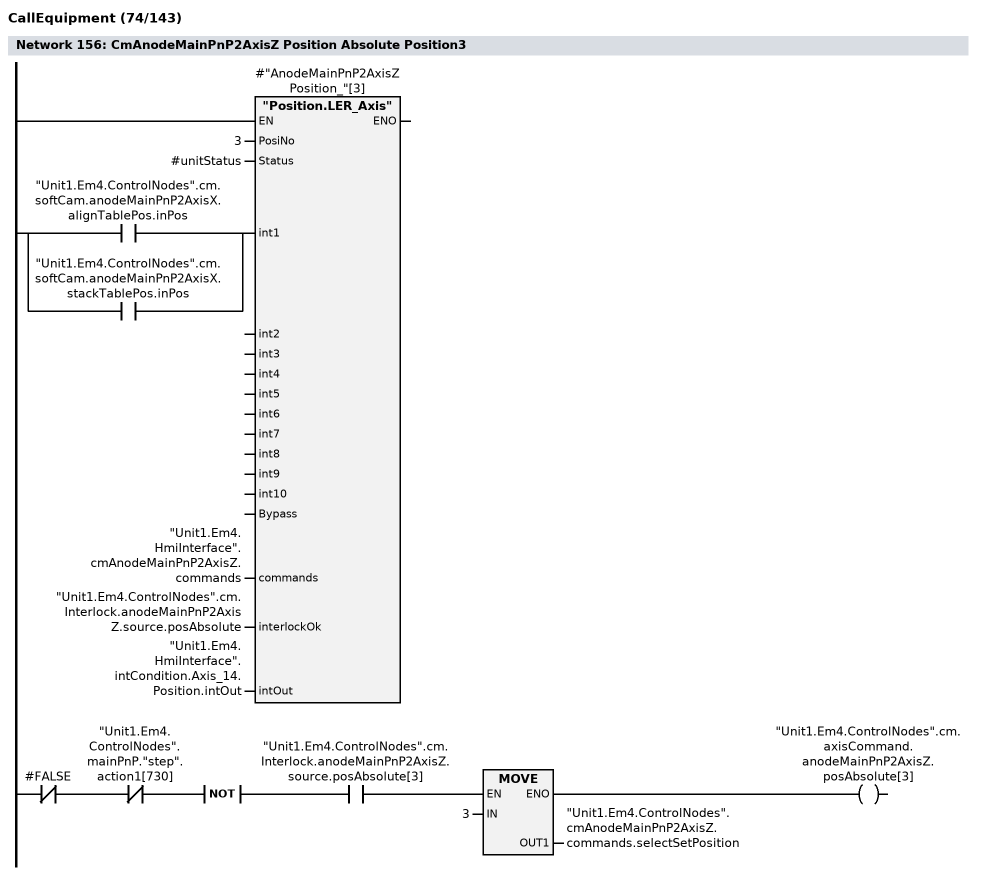
   RUNG wire#powerrail
      #"AnodeMainPnP2AxisZ Position_"[3](int1 := wire#w1, PosiNo := 3, Status := #unitStatus, int2 :=, int3 :=, int4 :=, int5 :=, int6 :=, int7 :=, int8 :=, int9 :=, int10 :=, Bypass :=, commands := "Unit1.Em4.HmiInterface".cmAnodeMainPnP2AxisZ.commands, interlockOk := "Unit1.Em4.ControlNodes".cm.Interlock.anodeMainPnP2AxisZ.source.posAbsolute, intOut := "Unit1.Em4.HmiInterface".intCondition.Axis_14.Position.intOut)
   END_RUNG
   RUNG wire#powerrail
      Contact( "Unit1.Em4.ControlNodes".cm.softCam.anodeMainPnP2AxisX.alignTablePos.inPos )
   END_RUNG wire#w1
   RUNG wire#powerrail
      Contact( "Unit1.Em4.ControlNodes".cm.softCam.anodeMainPnP2AxisX.stackTablePos.inPos )
   END_RUNG wire#w1
   RUNG wire#powerrail
      I_Contact( #FALSE )
      I_Contact( "Unit1.Em4.ControlNodes".mainPnP."step".action1[730] )
      Not()
      Contact( "Unit1.Em4.ControlNodes".cm.Interlock.anodeMainPnP2AxisZ.source.posAbsolute[3] )
      Move(in := 3, out1 => "Unit1.Em4.ControlNodes".cmAnodeMainPnP2AxisZ.commands.selectSetPosition)
      Coil( "Unit1.Em4.ControlNodes".cm.axisCommand.anodeMainPnP2AxisZ.posAbsolute[3] )
   END_RUNG
   // the same network as SCL:
   #"AnodeMainPnP2AxisZ Position_"[3](PosiNo := 3,   // "Position.LER_Axis"
                           Status := #unitStatus,
                           int1 := "Unit1.Em4.ControlNodes".cm.softCam.anodeMainPnP2AxisX.alignTablePos.inPos OR "Unit1.Em4.ControlNodes".cm.softCam.anodeMainPnP2AxisX.stackTablePos.inPos,
                           commands := "Unit1.Em4.HmiInterface".cmAnodeMainPnP2AxisZ.commands,
                           interlockOk := "Unit1.Em4.ControlNodes".cm.Interlock.anodeMainPnP2AxisZ.source.posAbsolute,
                           intOut := "Unit1.Em4.HmiInterface".intCondition.Axis_14.Position.intOut);
   #_w1 := NOT (NOT #FALSE AND NOT "Unit1.Em4.ControlNodes".mainPnP."step".action1[730]) AND "Unit1.Em4.ControlNodes".cm.Interlock.anodeMainPnP2AxisZ.source.posAbsolute[3];
   IF #_w1 THEN "Unit1.Em4.ControlNodes".cmAnodeMainPnP2AxisZ.commands.selectSetPosition := 3; END_IF;
   "Unit1.Em4.ControlNodes".cm.axisCommand.anodeMainPnP2AxisZ.posAbsolute[3] := #_w1;
END_REGION

REGION Network 157: CmAnodeMainPnP2AxisZ Position Absolute Position4
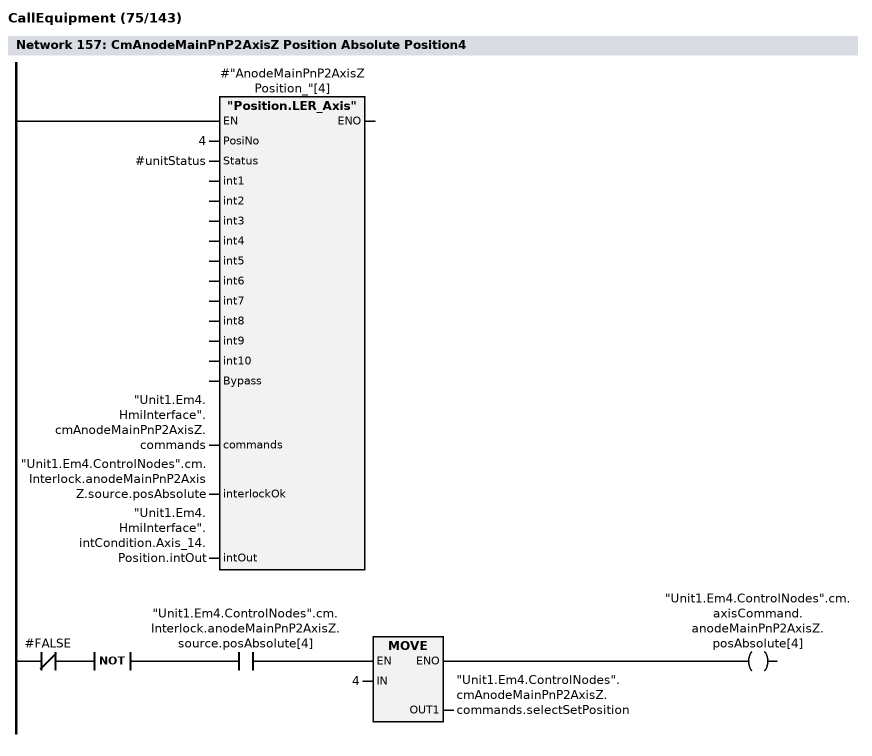
   RUNG wire#powerrail
      #"AnodeMainPnP2AxisZ Position_"[4](PosiNo := 4, Status := #unitStatus, int1 :=, int2 :=, int3 :=, int4 :=, int5 :=, int6 :=, int7 :=, int8 :=, int9 :=, int10 :=, Bypass :=, commands := "Unit1.Em4.HmiInterface".cmAnodeMainPnP2AxisZ.commands, interlockOk := "Unit1.Em4.ControlNodes".cm.Interlock.anodeMainPnP2AxisZ.source.posAbsolute, intOut := "Unit1.Em4.HmiInterface".intCondition.Axis_14.Position.intOut)
   END_RUNG
   RUNG wire#powerrail
      I_Contact( #FALSE )
      Not()
      Contact( "Unit1.Em4.ControlNodes".cm.Interlock.anodeMainPnP2AxisZ.source.posAbsolute[4] )
      Move(in := 4, out1 => "Unit1.Em4.ControlNodes".cmAnodeMainPnP2AxisZ.commands.selectSetPosition)
      Coil( "Unit1.Em4.ControlNodes".cm.axisCommand.anodeMainPnP2AxisZ.posAbsolute[4] )
   END_RUNG
   // the same network as SCL:
   #"AnodeMainPnP2AxisZ Position_"[4](PosiNo := 4,   // "Position.LER_Axis"
                           Status := #unitStatus,
                           commands := "Unit1.Em4.HmiInterface".cmAnodeMainPnP2AxisZ.commands,
                           interlockOk := "Unit1.Em4.ControlNodes".cm.Interlock.anodeMainPnP2AxisZ.source.posAbsolute,
                           intOut := "Unit1.Em4.HmiInterface".intCondition.Axis_14.Position.intOut);
   #_w1 := NOT (NOT #FALSE) AND "Unit1.Em4.ControlNodes".cm.Interlock.anodeMainPnP2AxisZ.source.posAbsolute[4];
   IF #_w1 THEN "Unit1.Em4.ControlNodes".cmAnodeMainPnP2AxisZ.commands.selectSetPosition := 4; END_IF;
   "Unit1.Em4.ControlNodes".cm.axisCommand.anodeMainPnP2AxisZ.posAbsolute[4] := #_w1;
END_REGION

REGION Network 158: CmAnodeMainPnP2AxisZ Position Absolute Position5
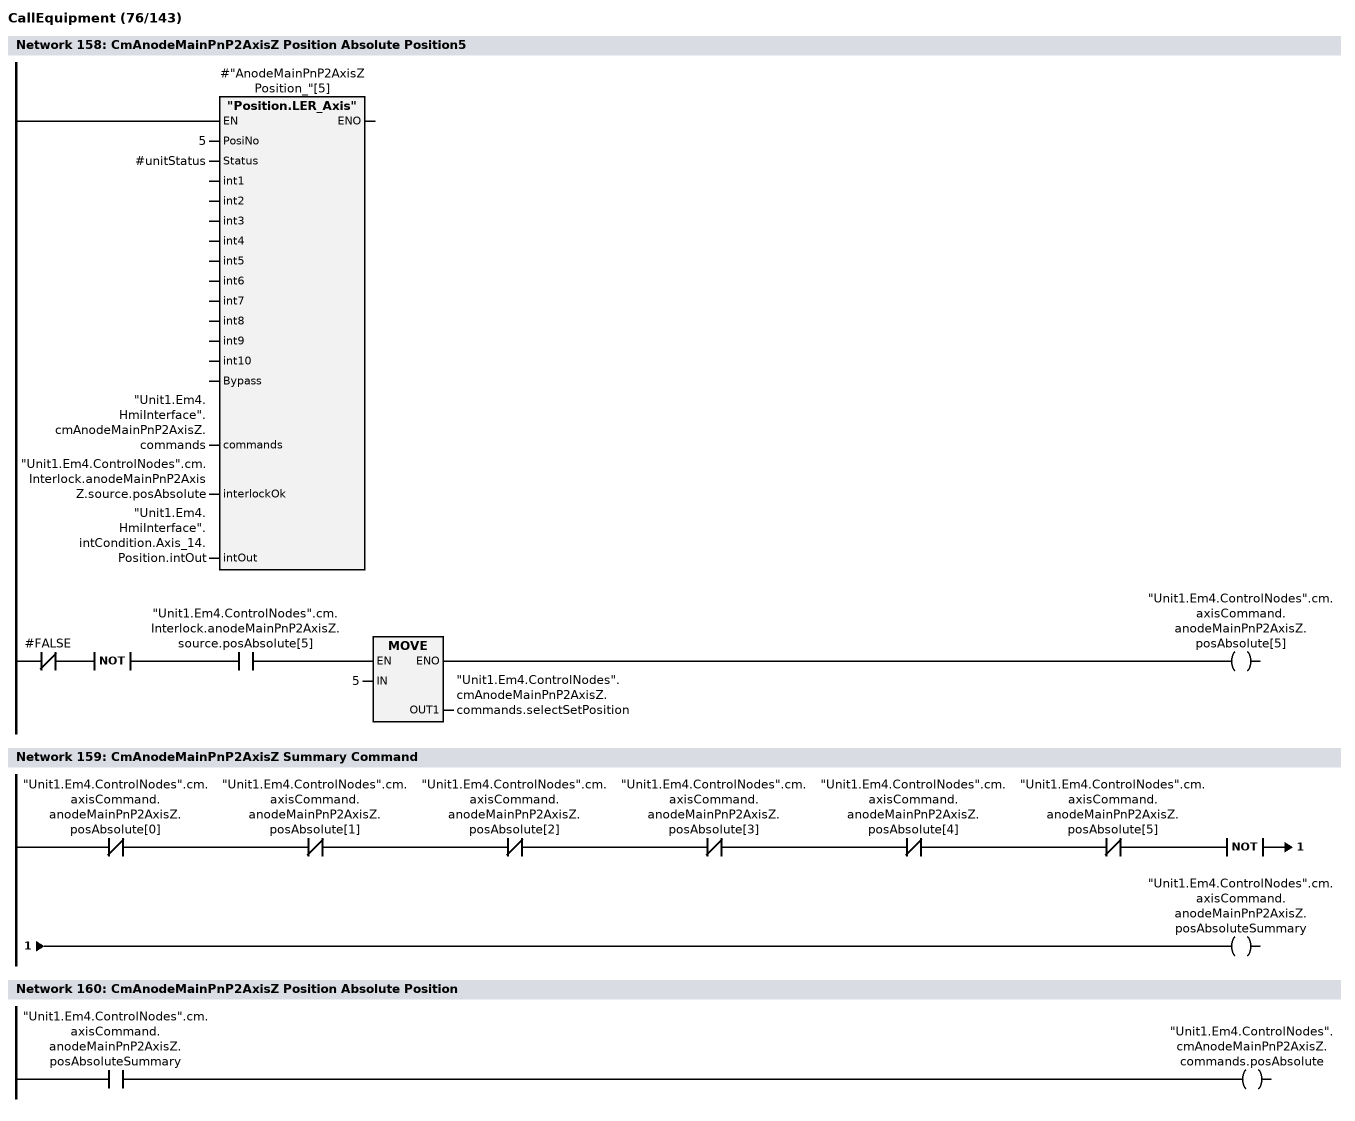
   RUNG wire#powerrail
      #"AnodeMainPnP2AxisZ Position_"[5](PosiNo := 5, Status := #unitStatus, int1 :=, int2 :=, int3 :=, int4 :=, int5 :=, int6 :=, int7 :=, int8 :=, int9 :=, int10 :=, Bypass :=, commands := "Unit1.Em4.HmiInterface".cmAnodeMainPnP2AxisZ.commands, interlockOk := "Unit1.Em4.ControlNodes".cm.Interlock.anodeMainPnP2AxisZ.source.posAbsolute, intOut := "Unit1.Em4.HmiInterface".intCondition.Axis_14.Position.intOut)
   END_RUNG
   RUNG wire#powerrail
      I_Contact( #FALSE )
      Not()
      Contact( "Unit1.Em4.ControlNodes".cm.Interlock.anodeMainPnP2AxisZ.source.posAbsolute[5] )
      Move(in := 5, out1 => "Unit1.Em4.ControlNodes".cmAnodeMainPnP2AxisZ.commands.selectSetPosition)
      Coil( "Unit1.Em4.ControlNodes".cm.axisCommand.anodeMainPnP2AxisZ.posAbsolute[5] )
   END_RUNG
   // the same network as SCL:
   #"AnodeMainPnP2AxisZ Position_"[5](PosiNo := 5,   // "Position.LER_Axis"
                           Status := #unitStatus,
                           commands := "Unit1.Em4.HmiInterface".cmAnodeMainPnP2AxisZ.commands,
                           interlockOk := "Unit1.Em4.ControlNodes".cm.Interlock.anodeMainPnP2AxisZ.source.posAbsolute,
                           intOut := "Unit1.Em4.HmiInterface".intCondition.Axis_14.Position.intOut);
   #_w1 := NOT (NOT #FALSE) AND "Unit1.Em4.ControlNodes".cm.Interlock.anodeMainPnP2AxisZ.source.posAbsolute[5];
   IF #_w1 THEN "Unit1.Em4.ControlNodes".cmAnodeMainPnP2AxisZ.commands.selectSetPosition := 5; END_IF;
   "Unit1.Em4.ControlNodes".cm.axisCommand.anodeMainPnP2AxisZ.posAbsolute[5] := #_w1;
END_REGION

REGION Network 159: CmAnodeMainPnP2AxisZ Summary Command
   RUNG wire#powerrail
      I_Contact( "Unit1.Em4.ControlNodes".cm.axisCommand.anodeMainPnP2AxisZ.posAbsolute[0] )
      I_Contact( "Unit1.Em4.ControlNodes".cm.axisCommand.anodeMainPnP2AxisZ.posAbsolute[1] )
      I_Contact( "Unit1.Em4.ControlNodes".cm.axisCommand.anodeMainPnP2AxisZ.posAbsolute[2] )
      I_Contact( "Unit1.Em4.ControlNodes".cm.axisCommand.anodeMainPnP2AxisZ.posAbsolute[3] )
      I_Contact( "Unit1.Em4.ControlNodes".cm.axisCommand.anodeMainPnP2AxisZ.posAbsolute[4] )
      I_Contact( "Unit1.Em4.ControlNodes".cm.axisCommand.anodeMainPnP2AxisZ.posAbsolute[5] )
      Not()
      Coil( "Unit1.Em4.ControlNodes".cm.axisCommand.anodeMainPnP2AxisZ.posAbsoluteSummary )
   END_RUNG
   // the same network as SCL:
   "Unit1.Em4.ControlNodes".cm.axisCommand.anodeMainPnP2AxisZ.posAbsoluteSummary := NOT (NOT "Unit1.Em4.ControlNodes".cm.axisCommand.anodeMainPnP2AxisZ.posAbsolute[0] AND NOT "Unit1.Em4.ControlNodes".cm.axisCommand.anodeMainPnP2AxisZ.posAbsolute[1] AND NOT "Unit1.Em4.ControlNodes".cm.axisCommand.anodeMainPnP2AxisZ.posAbsolute[2] AND NOT "Unit1.Em4.ControlNodes".cm.axisCommand.anodeMainPnP2AxisZ.posAbsolute[3] AND NOT "Unit1.Em4.ControlNodes".cm.axisCommand.anodeMainPnP2AxisZ.posAbsolute[4] AND NOT "Unit1.Em4.ControlNodes".cm.axisCommand.anodeMainPnP2AxisZ.posAbsolute[5]);
END_REGION

REGION Network 160: CmAnodeMainPnP2AxisZ Position Absolute Position
   RUNG wire#powerrail
      Contact( "Unit1.Em4.ControlNodes".cm.axisCommand.anodeMainPnP2AxisZ.posAbsoluteSummary )
      Coil( "Unit1.Em4.ControlNodes".cmAnodeMainPnP2AxisZ.commands.posAbsolute )
   END_RUNG
   // the same network as SCL:
   "Unit1.Em4.ControlNodes".cmAnodeMainPnP2AxisZ.commands.posAbsolute := "Unit1.Em4.ControlNodes".cm.axisCommand.anodeMainPnP2AxisZ.posAbsoluteSummary;
END_REGION

REGION Network 161: CmAnodeMainPnP1AxisZ Interlock Summary
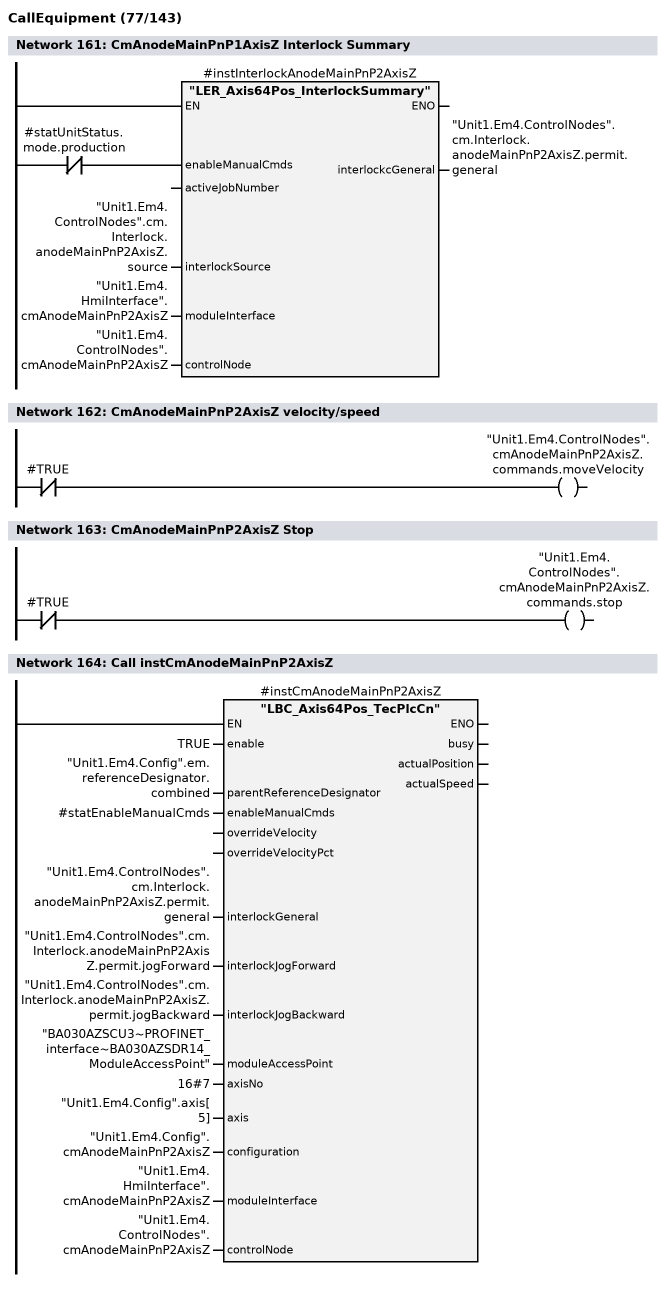
   RUNG wire#powerrail
      #instInterlockAnodeMainPnP2AxisZ(enableManualCmds := wire#w1, activeJobNumber :=, interlockSource := "Unit1.Em4.ControlNodes".cm.Interlock.anodeMainPnP2AxisZ.source, moduleInterface := "Unit1.Em4.HmiInterface".cmAnodeMainPnP2AxisZ, controlNode := "Unit1.Em4.ControlNodes".cmAnodeMainPnP2AxisZ, interlockcGeneral => "Unit1.Em4.ControlNodes".cm.Interlock.anodeMainPnP2AxisZ.permit.general)
   END_RUNG
   RUNG wire#powerrail
      I_Contact( #statUnitStatus.mode.production )
   END_RUNG wire#w1
   // the same network as SCL:
   #instInterlockAnodeMainPnP2AxisZ(enableManualCmds := NOT #statUnitStatus.mode.production,   // "LER_Axis64Pos_InterlockSummary"
                           interlockSource := "Unit1.Em4.ControlNodes".cm.Interlock.anodeMainPnP2AxisZ.source,
                           moduleInterface := "Unit1.Em4.HmiInterface".cmAnodeMainPnP2AxisZ,
                           controlNode := "Unit1.Em4.ControlNodes".cmAnodeMainPnP2AxisZ,
                           interlockcGeneral => "Unit1.Em4.ControlNodes".cm.Interlock.anodeMainPnP2AxisZ.permit.general);
END_REGION

REGION Network 162: CmAnodeMainPnP2AxisZ velocity/speed
   RUNG wire#powerrail
      I_Contact( #TRUE )
      Coil( "Unit1.Em4.ControlNodes".cmAnodeMainPnP2AxisZ.commands.moveVelocity )
   END_RUNG
   // the same network as SCL:
   "Unit1.Em4.ControlNodes".cmAnodeMainPnP2AxisZ.commands.moveVelocity := NOT #TRUE;
END_REGION

REGION Network 163: CmAnodeMainPnP2AxisZ Stop
   RUNG wire#powerrail
      I_Contact( #TRUE )
      Coil( "Unit1.Em4.ControlNodes".cmAnodeMainPnP2AxisZ.commands.stop )
   END_RUNG
   // the same network as SCL:
   "Unit1.Em4.ControlNodes".cmAnodeMainPnP2AxisZ.commands.stop := NOT #TRUE;
END_REGION

REGION Network 164: Call instCmAnodeMainPnP2AxisZ
   RUNG wire#powerrail
      #instCmAnodeMainPnP2AxisZ(enable := TRUE, parentReferenceDesignator := "Unit1.Em4.Config".em.referenceDesignator.combined, enableManualCmds := #statEnableManualCmds, overrideVelocity :=, overrideVelocityPct :=, interlockGeneral := "Unit1.Em4.ControlNodes".cm.Interlock.anodeMainPnP2AxisZ.permit.general, interlockJogForward := "Unit1.Em4.ControlNodes".cm.Interlock.anodeMainPnP2AxisZ.permit.jogForward, interlockJogBackward := "Unit1.Em4.ControlNodes".cm.Interlock.anodeMainPnP2AxisZ.permit.jogBackward, moduleAccessPoint := "BA030AZSCU3~PROFINET_interface~BA030AZSDR14_ModuleAccessPoint", axisNo := 16#7, axis := "Unit1.Em4.Config".axis[5], configuration := "Unit1.Em4.Config".cmAnodeMainPnP2AxisZ, moduleInterface := "Unit1.Em4.HmiInterface".cmAnodeMainPnP2AxisZ, controlNode := "Unit1.Em4.ControlNodes".cmAnodeMainPnP2AxisZ, busy =>, actualPosition =>, actualSpeed =>)
   END_RUNG
   // the same network as SCL:
   #instCmAnodeMainPnP2AxisZ(enable := TRUE,   // "LBC_Axis64Pos_TecPlcCn"
                           parentReferenceDesignator := "Unit1.Em4.Config".em.referenceDesignator.combined,
                           enableManualCmds := #statEnableManualCmds,
                           interlockGeneral := "Unit1.Em4.ControlNodes".cm.Interlock.anodeMainPnP2AxisZ.permit.general,
                           interlockJogForward := "Unit1.Em4.ControlNodes".cm.Interlock.anodeMainPnP2AxisZ.permit.jogForward,
                           interlockJogBackward := "Unit1.Em4.ControlNodes".cm.Interlock.anodeMainPnP2AxisZ.permit.jogBackward,
                           moduleAccessPoint := "BA030AZSCU3~PROFINET_interface~BA030AZSDR14_ModuleAccessPoint",
                           axisNo := 16#7,
                           axis := "Unit1.Em4.Config".axis[5],
                           configuration := "Unit1.Em4.Config".cmAnodeMainPnP2AxisZ,
                           moduleInterface := "Unit1.Em4.HmiInterface".cmAnodeMainPnP2AxisZ,
                           controlNode := "Unit1.Em4.ControlNodes".cmAnodeMainPnP2AxisZ);
END_REGION

REGION Network 165: CmAnodeMainPnP2AxisY SoftCam
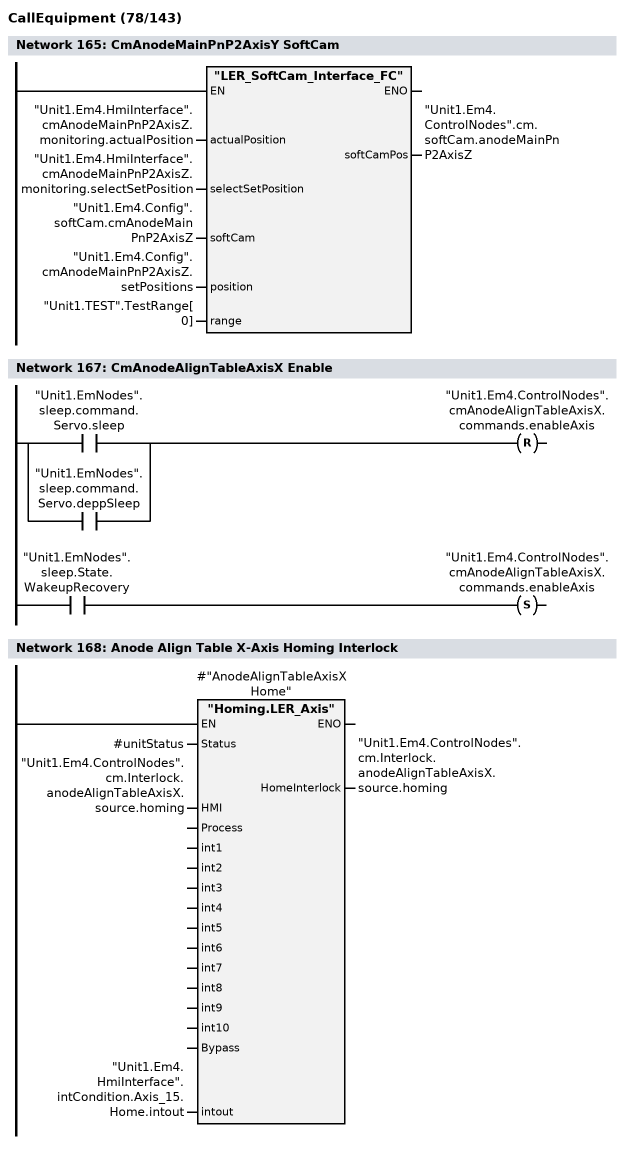
   RUNG wire#powerrail
      "LER_SoftCam_Interface_FC"(actualPosition := "Unit1.Em4.HmiInterface".cmAnodeMainPnP2AxisZ.monitoring.actualPosition, selectSetPosition := "Unit1.Em4.HmiInterface".cmAnodeMainPnP2AxisZ.monitoring.selectSetPosition, softCam := "Unit1.Em4.Config".softCam.cmAnodeMainPnP2AxisZ, position := "Unit1.Em4.Config".cmAnodeMainPnP2AxisZ.setPositions, range := "Unit1.TEST".TestRange[0], softCamPos => "Unit1.Em4.ControlNodes".cm.softCam.anodeMainPnP2AxisZ)
   END_RUNG
   // the same network as SCL:
   "LER_SoftCam_Interface_FC"(actualPosition := "Unit1.Em4.HmiInterface".cmAnodeMainPnP2AxisZ.monitoring.actualPosition,
                           selectSetPosition := "Unit1.Em4.HmiInterface".cmAnodeMainPnP2AxisZ.monitoring.selectSetPosition,
                           softCam := "Unit1.Em4.Config".softCam.cmAnodeMainPnP2AxisZ,
                           position := "Unit1.Em4.Config".cmAnodeMainPnP2AxisZ.setPositions,
                           range := "Unit1.TEST".TestRange[0],
                           softCamPos => "Unit1.Em4.ControlNodes".cm.softCam.anodeMainPnP2AxisZ);
END_REGION

REGION Network 167: CmAnodeAlignTableAxisX Enable
   RUNG wire#powerrail
      Contact( "Unit1.EmNodes".sleep.command.Servo.sleep )
      wire#w1
      R_Coil( "Unit1.Em4.ControlNodes".cmAnodeAlignTableAxisX.commands.enableAxis )
   END_RUNG
   RUNG wire#powerrail
      Contact( "Unit1.EmNodes".sleep.command.Servo.deppSleep )
   END_RUNG wire#w1
   RUNG wire#powerrail
      Contact( "Unit1.EmNodes".sleep.State.WakeupRecovery )
      S_Coil( "Unit1.Em4.ControlNodes".cmAnodeAlignTableAxisX.commands.enableAxis )
   END_RUNG
   // the same network as SCL:
   IF "Unit1.EmNodes".sleep.command.Servo.sleep OR "Unit1.EmNodes".sleep.command.Servo.deppSleep THEN
       "Unit1.Em4.ControlNodes".cmAnodeAlignTableAxisX.commands.enableAxis := FALSE;
   END_IF;
   IF "Unit1.EmNodes".sleep.State.WakeupRecovery THEN
       "Unit1.Em4.ControlNodes".cmAnodeAlignTableAxisX.commands.enableAxis := TRUE;
   END_IF;
END_REGION

REGION Network 168: Anode Align Table X-Axis Homing Interlock
   RUNG wire#powerrail
      #"AnodeAlignTableAxisX Home"(Status := #unitStatus, HMI := "Unit1.Em4.ControlNodes".cm.Interlock.anodeAlignTableAxisX.source.homing, Process :=, int1 :=, int2 :=, int3 :=, int4 :=, int5 :=, int6 :=, int7 :=, int8 :=, int9 :=, int10 :=, Bypass :=, intout := "Unit1.Em4.HmiInterface".intCondition.Axis_15.Home.intout, HomeInterlock => "Unit1.Em4.ControlNodes".cm.Interlock.anodeAlignTableAxisX.source.homing)
   END_RUNG
   // the same network as SCL:
   #"AnodeAlignTableAxisX Home"(Status := #unitStatus,   // "Homing.LER_Axis"
                           HMI := "Unit1.Em4.ControlNodes".cm.Interlock.anodeAlignTableAxisX.source.homing,
                           intout := "Unit1.Em4.HmiInterface".intCondition.Axis_15.Home.intout,
                           HomeInterlock => "Unit1.Em4.ControlNodes".cm.Interlock.anodeAlignTableAxisX.source.homing);
END_REGION

REGION Network 169: CmAnodeAlignTableAxisX Position Absolute Jog
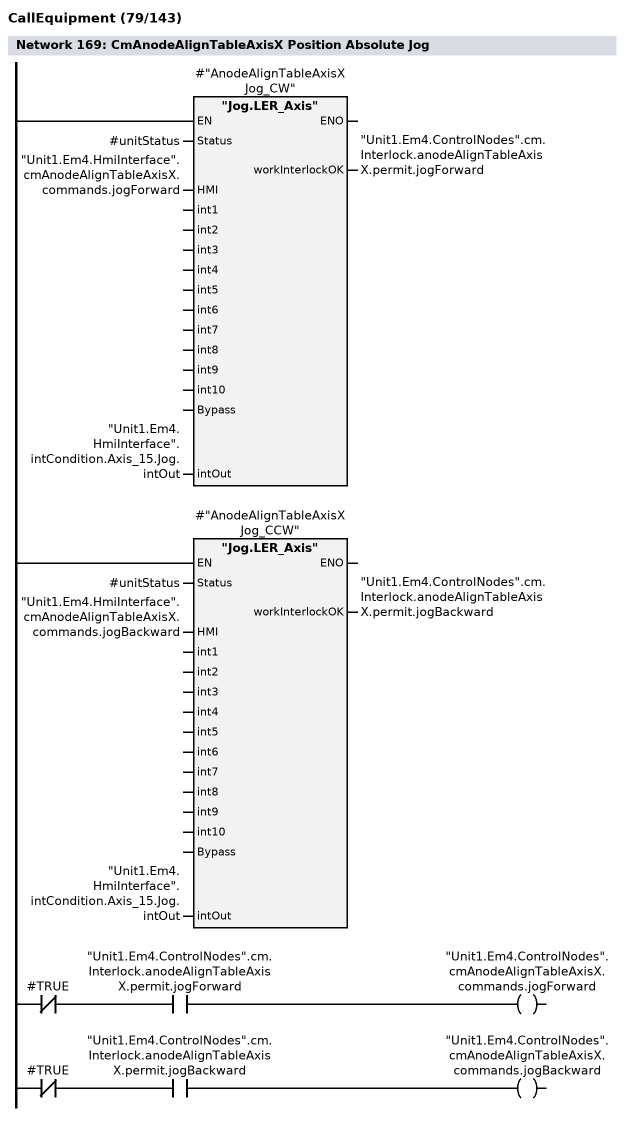
   RUNG wire#powerrail
      #"AnodeAlignTableAxisX Jog_CW"(Status := #unitStatus, HMI := "Unit1.Em4.HmiInterface".cmAnodeAlignTableAxisX.commands.jogForward, int1 :=, int2 :=, int3 :=, int4 :=, int5 :=, int6 :=, int7 :=, int8 :=, int9 :=, int10 :=, Bypass :=, intOut := "Unit1.Em4.HmiInterface".intCondition.Axis_15.Jog.intOut, workInterlockOK => "Unit1.Em4.ControlNodes".cm.Interlock.anodeAlignTableAxisX.permit.jogForward)
   END_RUNG
   RUNG wire#powerrail
      #"AnodeAlignTableAxisX Jog_CCW"(Status := #unitStatus, HMI := "Unit1.Em4.HmiInterface".cmAnodeAlignTableAxisX.commands.jogBackward, int1 :=, int2 :=, int3 :=, int4 :=, int5 :=, int6 :=, int7 :=, int8 :=, int9 :=, int10 :=, Bypass :=, intOut := "Unit1.Em4.HmiInterface".intCondition.Axis_15.Jog.intOut, workInterlockOK => "Unit1.Em4.ControlNodes".cm.Interlock.anodeAlignTableAxisX.permit.jogBackward)
   END_RUNG
   RUNG wire#powerrail
      I_Contact( #TRUE )
      Contact( "Unit1.Em4.ControlNodes".cm.Interlock.anodeAlignTableAxisX.permit.jogForward )
      Coil( "Unit1.Em4.ControlNodes".cmAnodeAlignTableAxisX.commands.jogForward )
   END_RUNG
   RUNG wire#powerrail
      I_Contact( #TRUE )
      Contact( "Unit1.Em4.ControlNodes".cm.Interlock.anodeAlignTableAxisX.permit.jogBackward )
      Coil( "Unit1.Em4.ControlNodes".cmAnodeAlignTableAxisX.commands.jogBackward )
   END_RUNG
   // the same network as SCL:
   #"AnodeAlignTableAxisX Jog_CW"(Status := #unitStatus,   // "Jog.LER_Axis"
                           HMI := "Unit1.Em4.HmiInterface".cmAnodeAlignTableAxisX.commands.jogForward,
                           intOut := "Unit1.Em4.HmiInterface".intCondition.Axis_15.Jog.intOut,
                           workInterlockOK => "Unit1.Em4.ControlNodes".cm.Interlock.anodeAlignTableAxisX.permit.jogForward);
   #"AnodeAlignTableAxisX Jog_CCW"(Status := #unitStatus,   // "Jog.LER_Axis"
                           HMI := "Unit1.Em4.HmiInterface".cmAnodeAlignTableAxisX.commands.jogBackward,
                           intOut := "Unit1.Em4.HmiInterface".intCondition.Axis_15.Jog.intOut,
                           workInterlockOK => "Unit1.Em4.ControlNodes".cm.Interlock.anodeAlignTableAxisX.permit.jogBackward);
   "Unit1.Em4.ControlNodes".cmAnodeAlignTableAxisX.commands.jogForward := NOT #TRUE AND "Unit1.Em4.ControlNodes".cm.Interlock.anodeAlignTableAxisX.permit.jogForward;
   "Unit1.Em4.ControlNodes".cmAnodeAlignTableAxisX.commands.jogBackward := NOT #TRUE AND "Unit1.Em4.ControlNodes".cm.Interlock.anodeAlignTableAxisX.permit.jogBackward;
END_REGION

REGION Network 170: CmAnodeAlignTableAxisX Position Absolute Position0
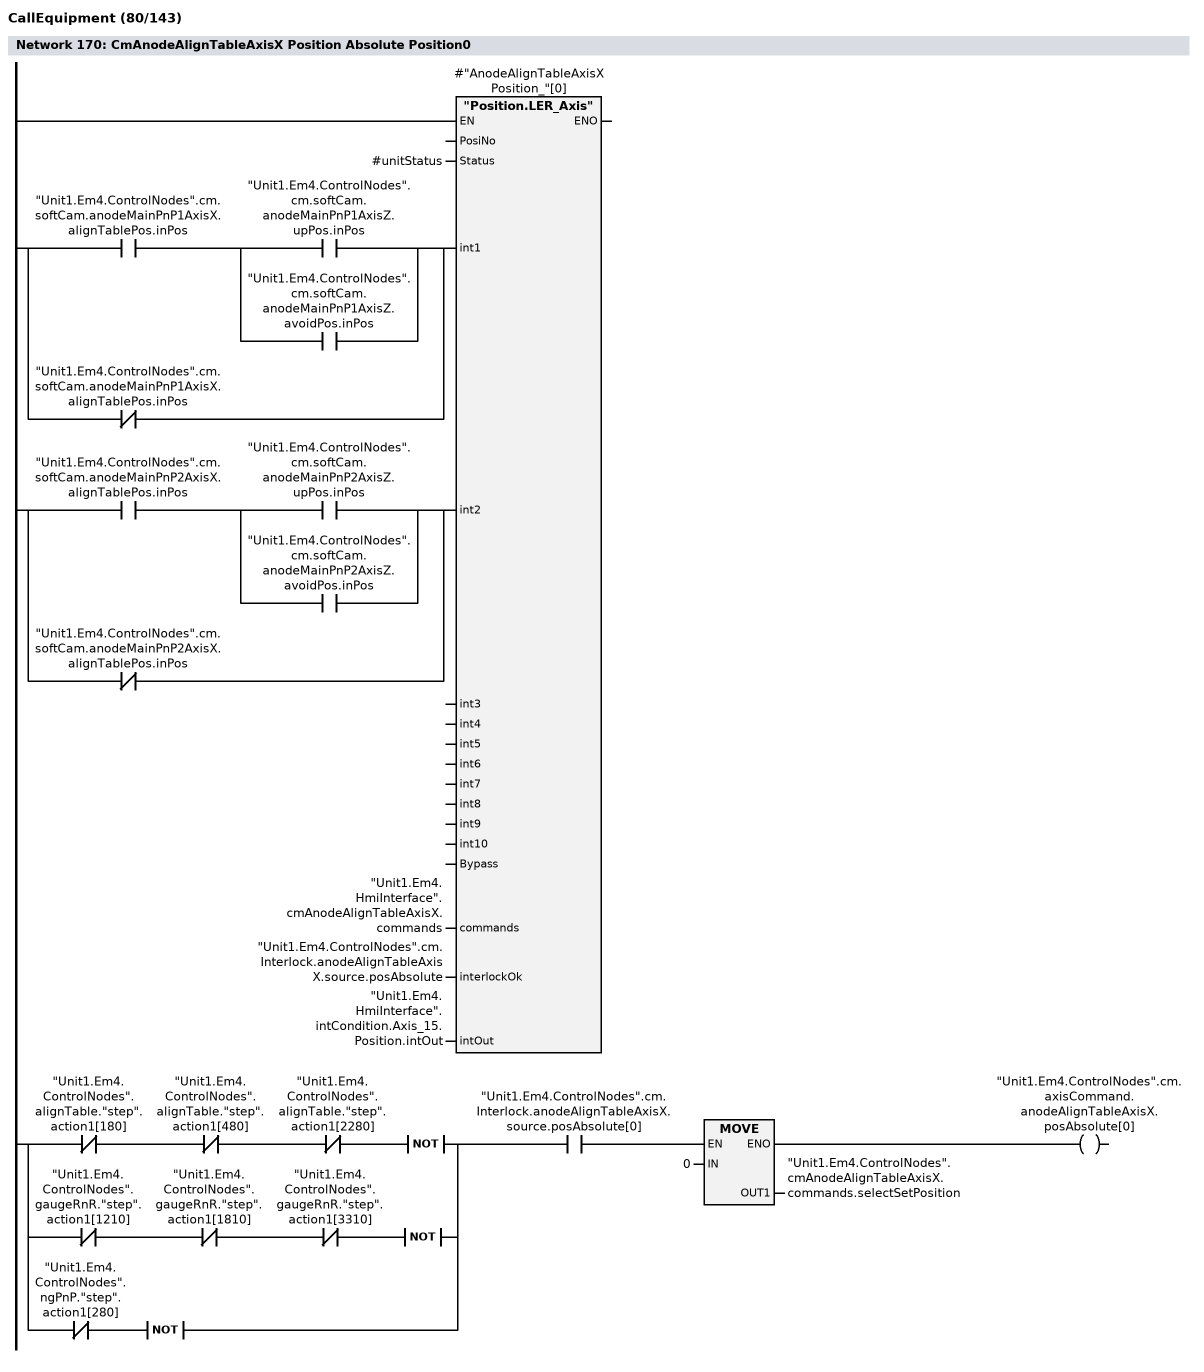
   RUNG wire#powerrail
      #"AnodeAlignTableAxisX Position_"[0](int1 := wire#w2, int2 := wire#w4, PosiNo :=, Status := #unitStatus, int3 :=, int4 :=, int5 :=, int6 :=, int7 :=, int8 :=, int9 :=, int10 :=, Bypass :=, commands := "Unit1.Em4.HmiInterface".cmAnodeAlignTableAxisX.commands, interlockOk := "Unit1.Em4.ControlNodes".cm.Interlock.anodeAlignTableAxisX.source.posAbsolute, intOut := "Unit1.Em4.HmiInterface".intCondition.Axis_15.Position.intOut)
   END_RUNG
   RUNG wire#powerrail
      Contact( "Unit1.Em4.ControlNodes".cm.softCam.anodeMainPnP1AxisX.alignTablePos.inPos )
      wire#w1
      Contact( "Unit1.Em4.ControlNodes".cm.softCam.anodeMainPnP1AxisZ.upPos.inPos )
   END_RUNG wire#w2
   RUNG wire#w1
      Contact( "Unit1.Em4.ControlNodes".cm.softCam.anodeMainPnP1AxisZ.avoidPos.inPos )
   END_RUNG wire#w2
   RUNG wire#powerrail
      I_Contact( "Unit1.Em4.ControlNodes".cm.softCam.anodeMainPnP1AxisX.alignTablePos.inPos )
   END_RUNG wire#w2
   RUNG wire#powerrail
      Contact( "Unit1.Em4.ControlNodes".cm.softCam.anodeMainPnP2AxisX.alignTablePos.inPos )
      wire#w3
      Contact( "Unit1.Em4.ControlNodes".cm.softCam.anodeMainPnP2AxisZ.upPos.inPos )
   END_RUNG wire#w4
   RUNG wire#w3
      Contact( "Unit1.Em4.ControlNodes".cm.softCam.anodeMainPnP2AxisZ.avoidPos.inPos )
   END_RUNG wire#w4
   RUNG wire#powerrail
      I_Contact( "Unit1.Em4.ControlNodes".cm.softCam.anodeMainPnP2AxisX.alignTablePos.inPos )
   END_RUNG wire#w4
   RUNG wire#powerrail
      I_Contact( "Unit1.Em4.ControlNodes".alignTable."step".action1[180] )
      I_Contact( "Unit1.Em4.ControlNodes".alignTable."step".action1[480] )
      I_Contact( "Unit1.Em4.ControlNodes".alignTable."step".action1[2280] )
      Not()
      wire#w5
      Contact( "Unit1.Em4.ControlNodes".cm.Interlock.anodeAlignTableAxisX.source.posAbsolute[0] )
      Move(in := 0, out1 => "Unit1.Em4.ControlNodes".cmAnodeAlignTableAxisX.commands.selectSetPosition)
      Coil( "Unit1.Em4.ControlNodes".cm.axisCommand.anodeAlignTableAxisX.posAbsolute[0] )
   END_RUNG
   RUNG wire#powerrail
      I_Contact( "Unit1.Em4.ControlNodes".gaugeRnR."step".action1[1210] )
      I_Contact( "Unit1.Em4.ControlNodes".gaugeRnR."step".action1[1810] )
      I_Contact( "Unit1.Em4.ControlNodes".gaugeRnR."step".action1[3310] )
      Not()
   END_RUNG wire#w5
   RUNG wire#powerrail
      I_Contact( "Unit1.Em4.ControlNodes".ngPnP."step".action1[280] )
      Not()
   END_RUNG wire#w5
   // the same network as SCL:
   #"AnodeAlignTableAxisX Position_"[0](Status := #unitStatus,   // "Position.LER_Axis"
                           int1 := ("Unit1.Em4.ControlNodes".cm.softCam.anodeMainPnP1AxisX.alignTablePos.inPos AND ("Unit1.Em4.ControlNodes".cm.softCam.anodeMainPnP1AxisZ.upPos.inPos OR "Unit1.Em4.ControlNodes".cm.softCam.anodeMainPnP1AxisZ.avoidPos.inPos)) OR NOT "Unit1.Em4.ControlNodes".cm.softCam.anodeMainPnP1AxisX.alignTablePos.inPos,
                           int2 := ("Unit1.Em4.ControlNodes".cm.softCam.anodeMainPnP2AxisX.alignTablePos.inPos AND ("Unit1.Em4.ControlNodes".cm.softCam.anodeMainPnP2AxisZ.upPos.inPos OR "Unit1.Em4.ControlNodes".cm.softCam.anodeMainPnP2AxisZ.avoidPos.inPos)) OR NOT "Unit1.Em4.ControlNodes".cm.softCam.anodeMainPnP2AxisX.alignTablePos.inPos,
                           commands := "Unit1.Em4.HmiInterface".cmAnodeAlignTableAxisX.commands,
                           interlockOk := "Unit1.Em4.ControlNodes".cm.Interlock.anodeAlignTableAxisX.source.posAbsolute,
                           intOut := "Unit1.Em4.HmiInterface".intCondition.Axis_15.Position.intOut);
   #_w1 := (NOT (NOT "Unit1.Em4.ControlNodes".alignTable."step".action1[180] AND NOT "Unit1.Em4.ControlNodes".alignTable."step".action1[480] AND NOT "Unit1.Em4.ControlNodes".alignTable."step".action1[2280]) OR NOT (NOT "Unit1.Em4.ControlNodes".gaugeRnR."step".action1[1210] AND NOT "Unit1.Em4.ControlNodes".gaugeRnR."step".action1[1810] AND NOT "Unit1.Em4.ControlNodes".gaugeRnR."step".action1[3310]) OR NOT (NOT "Unit1.Em4.ControlNodes".ngPnP."step".action1[280])) AND "Unit1.Em4.ControlNodes".cm.Interlock.anodeAlignTableAxisX.source.posAbsolute[0];
   IF #_w1 THEN "Unit1.Em4.ControlNodes".cmAnodeAlignTableAxisX.commands.selectSetPosition := 0; END_IF;
   "Unit1.Em4.ControlNodes".cm.axisCommand.anodeAlignTableAxisX.posAbsolute[0] := #_w1;
END_REGION

REGION Network 171: CmAnodeAlignTableAxisX Position Absolute Position1
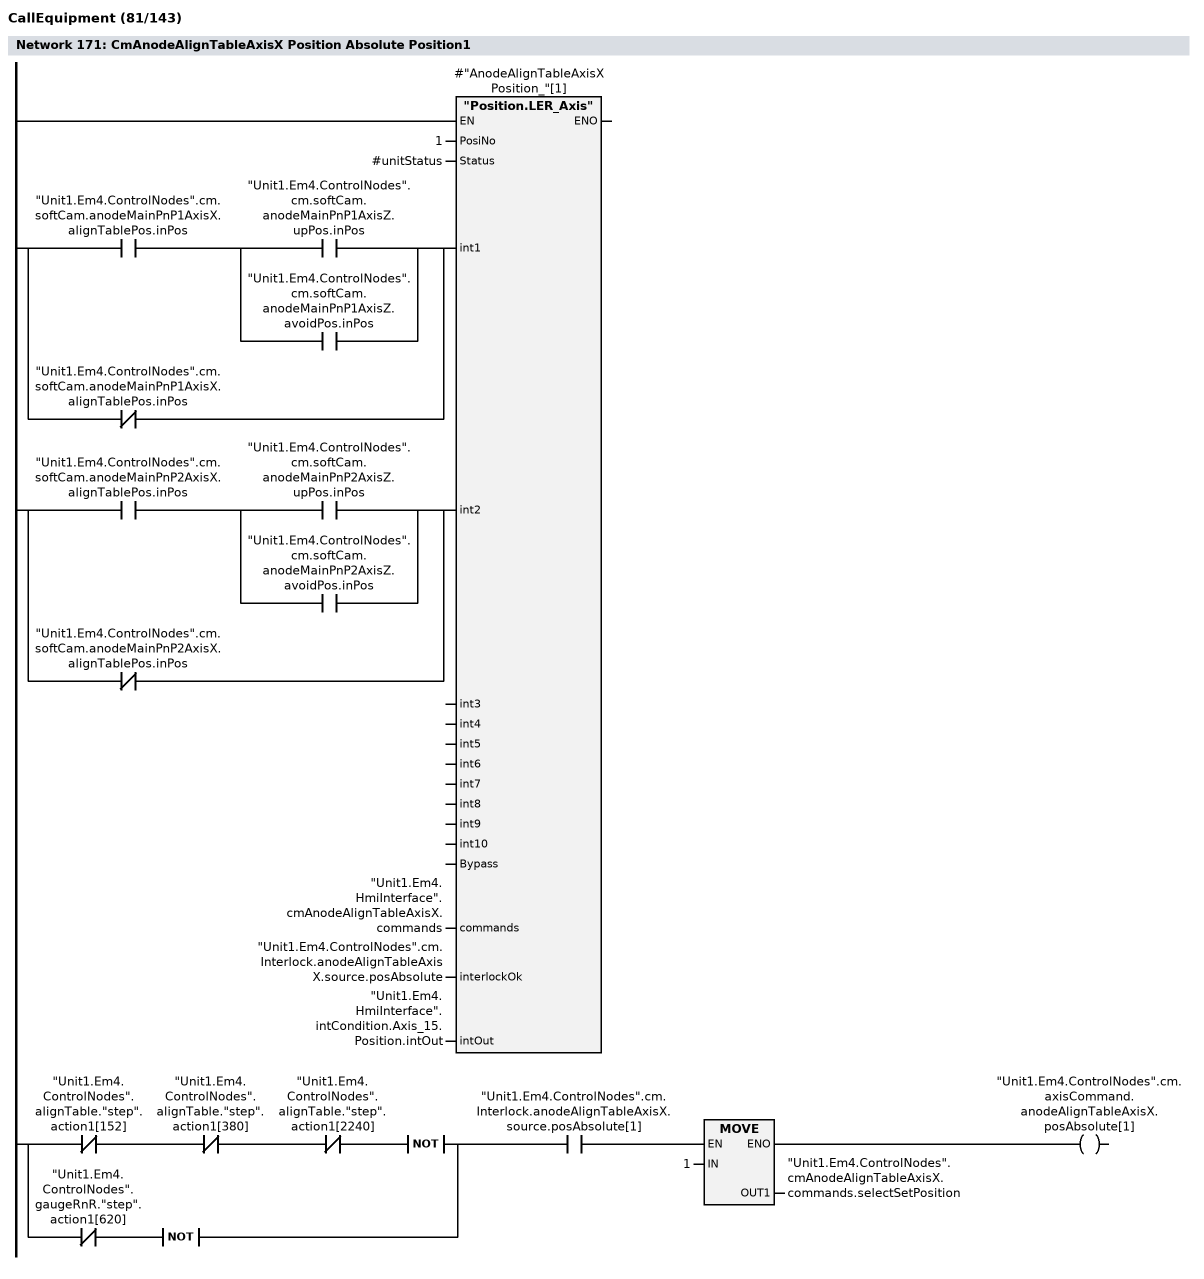
   RUNG wire#powerrail
      #"AnodeAlignTableAxisX Position_"[1](int1 := wire#w2, int2 := wire#w4, PosiNo := 1, Status := #unitStatus, int3 :=, int4 :=, int5 :=, int6 :=, int7 :=, int8 :=, int9 :=, int10 :=, Bypass :=, commands := "Unit1.Em4.HmiInterface".cmAnodeAlignTableAxisX.commands, interlockOk := "Unit1.Em4.ControlNodes".cm.Interlock.anodeAlignTableAxisX.source.posAbsolute, intOut := "Unit1.Em4.HmiInterface".intCondition.Axis_15.Position.intOut)
   END_RUNG
   RUNG wire#powerrail
      Contact( "Unit1.Em4.ControlNodes".cm.softCam.anodeMainPnP1AxisX.alignTablePos.inPos )
      wire#w1
      Contact( "Unit1.Em4.ControlNodes".cm.softCam.anodeMainPnP1AxisZ.upPos.inPos )
   END_RUNG wire#w2
   RUNG wire#w1
      Contact( "Unit1.Em4.ControlNodes".cm.softCam.anodeMainPnP1AxisZ.avoidPos.inPos )
   END_RUNG wire#w2
   RUNG wire#powerrail
      I_Contact( "Unit1.Em4.ControlNodes".cm.softCam.anodeMainPnP1AxisX.alignTablePos.inPos )
   END_RUNG wire#w2
   RUNG wire#powerrail
      Contact( "Unit1.Em4.ControlNodes".cm.softCam.anodeMainPnP2AxisX.alignTablePos.inPos )
      wire#w3
      Contact( "Unit1.Em4.ControlNodes".cm.softCam.anodeMainPnP2AxisZ.upPos.inPos )
   END_RUNG wire#w4
   RUNG wire#w3
      Contact( "Unit1.Em4.ControlNodes".cm.softCam.anodeMainPnP2AxisZ.avoidPos.inPos )
   END_RUNG wire#w4
   RUNG wire#powerrail
      I_Contact( "Unit1.Em4.ControlNodes".cm.softCam.anodeMainPnP2AxisX.alignTablePos.inPos )
   END_RUNG wire#w4
   RUNG wire#powerrail
      I_Contact( "Unit1.Em4.ControlNodes".alignTable."step".action1[152] )
      I_Contact( "Unit1.Em4.ControlNodes".alignTable."step".action1[380] )
      I_Contact( "Unit1.Em4.ControlNodes".alignTable."step".action1[2240] )
      Not()
      wire#w5
      Contact( "Unit1.Em4.ControlNodes".cm.Interlock.anodeAlignTableAxisX.source.posAbsolute[1] )
      Move(in := 1, out1 => "Unit1.Em4.ControlNodes".cmAnodeAlignTableAxisX.commands.selectSetPosition)
      Coil( "Unit1.Em4.ControlNodes".cm.axisCommand.anodeAlignTableAxisX.posAbsolute[1] )
   END_RUNG
   RUNG wire#powerrail
      I_Contact( "Unit1.Em4.ControlNodes".gaugeRnR."step".action1[620] )
      Not()
   END_RUNG wire#w5
   // the same network as SCL:
   #"AnodeAlignTableAxisX Position_"[1](PosiNo := 1,   // "Position.LER_Axis"
                           Status := #unitStatus,
                           int1 := ("Unit1.Em4.ControlNodes".cm.softCam.anodeMainPnP1AxisX.alignTablePos.inPos AND ("Unit1.Em4.ControlNodes".cm.softCam.anodeMainPnP1AxisZ.upPos.inPos OR "Unit1.Em4.ControlNodes".cm.softCam.anodeMainPnP1AxisZ.avoidPos.inPos)) OR NOT "Unit1.Em4.ControlNodes".cm.softCam.anodeMainPnP1AxisX.alignTablePos.inPos,
                           int2 := ("Unit1.Em4.ControlNodes".cm.softCam.anodeMainPnP2AxisX.alignTablePos.inPos AND ("Unit1.Em4.ControlNodes".cm.softCam.anodeMainPnP2AxisZ.upPos.inPos OR "Unit1.Em4.ControlNodes".cm.softCam.anodeMainPnP2AxisZ.avoidPos.inPos)) OR NOT "Unit1.Em4.ControlNodes".cm.softCam.anodeMainPnP2AxisX.alignTablePos.inPos,
                           commands := "Unit1.Em4.HmiInterface".cmAnodeAlignTableAxisX.commands,
                           interlockOk := "Unit1.Em4.ControlNodes".cm.Interlock.anodeAlignTableAxisX.source.posAbsolute,
                           intOut := "Unit1.Em4.HmiInterface".intCondition.Axis_15.Position.intOut);
   #_w1 := (NOT (NOT "Unit1.Em4.ControlNodes".alignTable."step".action1[152] AND NOT "Unit1.Em4.ControlNodes".alignTable."step".action1[380] AND NOT "Unit1.Em4.ControlNodes".alignTable."step".action1[2240]) OR NOT (NOT "Unit1.Em4.ControlNodes".gaugeRnR."step".action1[620])) AND "Unit1.Em4.ControlNodes".cm.Interlock.anodeAlignTableAxisX.source.posAbsolute[1];
   IF #_w1 THEN "Unit1.Em4.ControlNodes".cmAnodeAlignTableAxisX.commands.selectSetPosition := 1; END_IF;
   "Unit1.Em4.ControlNodes".cm.axisCommand.anodeAlignTableAxisX.posAbsolute[1] := #_w1;
END_REGION

REGION Network 172: CmAnodeAlignTableAxisX Position Absolute Position2
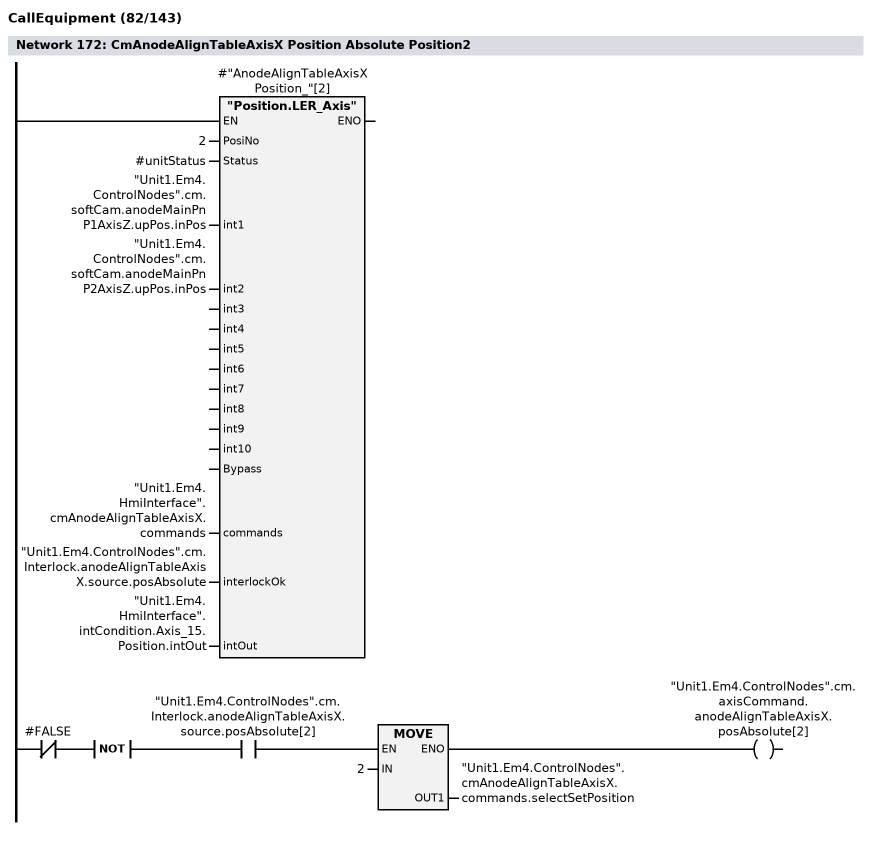
   RUNG wire#powerrail
      #"AnodeAlignTableAxisX Position_"[2](PosiNo := 2, Status := #unitStatus, int1 := "Unit1.Em4.ControlNodes".cm.softCam.anodeMainPnP1AxisZ.upPos.inPos, int2 := "Unit1.Em4.ControlNodes".cm.softCam.anodeMainPnP2AxisZ.upPos.inPos, int3 :=, int4 :=, int5 :=, int6 :=, int7 :=, int8 :=, int9 :=, int10 :=, Bypass :=, commands := "Unit1.Em4.HmiInterface".cmAnodeAlignTableAxisX.commands, interlockOk := "Unit1.Em4.ControlNodes".cm.Interlock.anodeAlignTableAxisX.source.posAbsolute, intOut := "Unit1.Em4.HmiInterface".intCondition.Axis_15.Position.intOut)
   END_RUNG
   RUNG wire#powerrail
      I_Contact( #FALSE )
      Not()
      Contact( "Unit1.Em4.ControlNodes".cm.Interlock.anodeAlignTableAxisX.source.posAbsolute[2] )
      Move(in := 2, out1 => "Unit1.Em4.ControlNodes".cmAnodeAlignTableAxisX.commands.selectSetPosition)
      Coil( "Unit1.Em4.ControlNodes".cm.axisCommand.anodeAlignTableAxisX.posAbsolute[2] )
   END_RUNG
   // the same network as SCL:
   #"AnodeAlignTableAxisX Position_"[2](PosiNo := 2,   // "Position.LER_Axis"
                           Status := #unitStatus,
                           int1 := "Unit1.Em4.ControlNodes".cm.softCam.anodeMainPnP1AxisZ.upPos.inPos,
                           int2 := "Unit1.Em4.ControlNodes".cm.softCam.anodeMainPnP2AxisZ.upPos.inPos,
                           commands := "Unit1.Em4.HmiInterface".cmAnodeAlignTableAxisX.commands,
                           interlockOk := "Unit1.Em4.ControlNodes".cm.Interlock.anodeAlignTableAxisX.source.posAbsolute,
                           intOut := "Unit1.Em4.HmiInterface".intCondition.Axis_15.Position.intOut);
   #_w1 := NOT (NOT #FALSE) AND "Unit1.Em4.ControlNodes".cm.Interlock.anodeAlignTableAxisX.source.posAbsolute[2];
   IF #_w1 THEN "Unit1.Em4.ControlNodes".cmAnodeAlignTableAxisX.commands.selectSetPosition := 2; END_IF;
   "Unit1.Em4.ControlNodes".cm.axisCommand.anodeAlignTableAxisX.posAbsolute[2] := #_w1;
END_REGION

REGION Network 173: CmAnodeAlignTableAxisX Position Absolute Position3
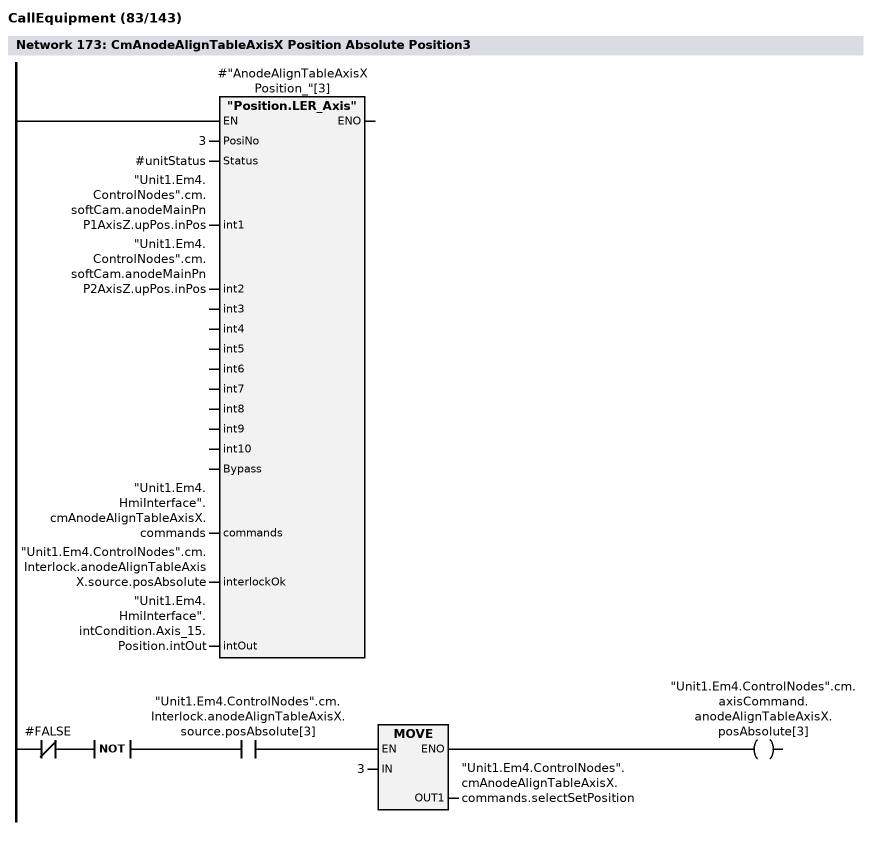
   RUNG wire#powerrail
      #"AnodeAlignTableAxisX Position_"[3](PosiNo := 3, Status := #unitStatus, int1 := "Unit1.Em4.ControlNodes".cm.softCam.anodeMainPnP1AxisZ.upPos.inPos, int2 := "Unit1.Em4.ControlNodes".cm.softCam.anodeMainPnP2AxisZ.upPos.inPos, int3 :=, int4 :=, int5 :=, int6 :=, int7 :=, int8 :=, int9 :=, int10 :=, Bypass :=, commands := "Unit1.Em4.HmiInterface".cmAnodeAlignTableAxisX.commands, interlockOk := "Unit1.Em4.ControlNodes".cm.Interlock.anodeAlignTableAxisX.source.posAbsolute, intOut := "Unit1.Em4.HmiInterface".intCondition.Axis_15.Position.intOut)
   END_RUNG
   RUNG wire#powerrail
      I_Contact( #FALSE )
      Not()
      Contact( "Unit1.Em4.ControlNodes".cm.Interlock.anodeAlignTableAxisX.source.posAbsolute[3] )
      Move(in := 3, out1 => "Unit1.Em4.ControlNodes".cmAnodeAlignTableAxisX.commands.selectSetPosition)
      Coil( "Unit1.Em4.ControlNodes".cm.axisCommand.anodeAlignTableAxisX.posAbsolute[3] )
   END_RUNG
   // the same network as SCL:
   #"AnodeAlignTableAxisX Position_"[3](PosiNo := 3,   // "Position.LER_Axis"
                           Status := #unitStatus,
                           int1 := "Unit1.Em4.ControlNodes".cm.softCam.anodeMainPnP1AxisZ.upPos.inPos,
                           int2 := "Unit1.Em4.ControlNodes".cm.softCam.anodeMainPnP2AxisZ.upPos.inPos,
                           commands := "Unit1.Em4.HmiInterface".cmAnodeAlignTableAxisX.commands,
                           interlockOk := "Unit1.Em4.ControlNodes".cm.Interlock.anodeAlignTableAxisX.source.posAbsolute,
                           intOut := "Unit1.Em4.HmiInterface".intCondition.Axis_15.Position.intOut);
   #_w1 := NOT (NOT #FALSE) AND "Unit1.Em4.ControlNodes".cm.Interlock.anodeAlignTableAxisX.source.posAbsolute[3];
   IF #_w1 THEN "Unit1.Em4.ControlNodes".cmAnodeAlignTableAxisX.commands.selectSetPosition := 3; END_IF;
   "Unit1.Em4.ControlNodes".cm.axisCommand.anodeAlignTableAxisX.posAbsolute[3] := #_w1;
END_REGION

REGION Network 174: CmAnodeAlignTableAxisX Position Absolute Position4
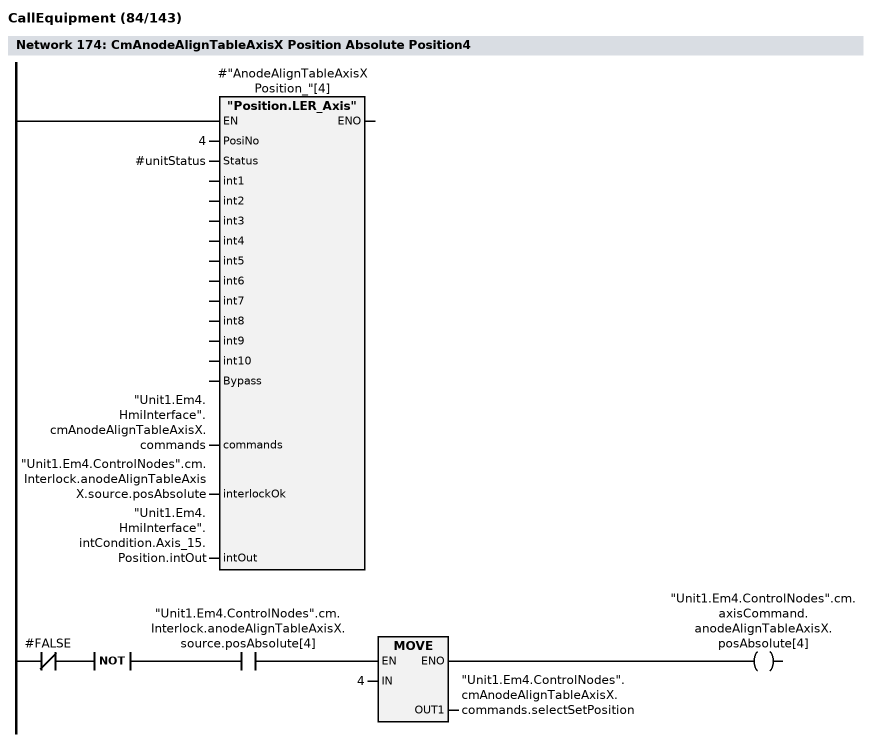
   RUNG wire#powerrail
      #"AnodeAlignTableAxisX Position_"[4](PosiNo := 4, Status := #unitStatus, int1 :=, int2 :=, int3 :=, int4 :=, int5 :=, int6 :=, int7 :=, int8 :=, int9 :=, int10 :=, Bypass :=, commands := "Unit1.Em4.HmiInterface".cmAnodeAlignTableAxisX.commands, interlockOk := "Unit1.Em4.ControlNodes".cm.Interlock.anodeAlignTableAxisX.source.posAbsolute, intOut := "Unit1.Em4.HmiInterface".intCondition.Axis_15.Position.intOut)
   END_RUNG
   RUNG wire#powerrail
      I_Contact( #FALSE )
      Not()
      Contact( "Unit1.Em4.ControlNodes".cm.Interlock.anodeAlignTableAxisX.source.posAbsolute[4] )
      Move(in := 4, out1 => "Unit1.Em4.ControlNodes".cmAnodeAlignTableAxisX.commands.selectSetPosition)
      Coil( "Unit1.Em4.ControlNodes".cm.axisCommand.anodeAlignTableAxisX.posAbsolute[4] )
   END_RUNG
   // the same network as SCL:
   #"AnodeAlignTableAxisX Position_"[4](PosiNo := 4,   // "Position.LER_Axis"
                           Status := #unitStatus,
                           commands := "Unit1.Em4.HmiInterface".cmAnodeAlignTableAxisX.commands,
                           interlockOk := "Unit1.Em4.ControlNodes".cm.Interlock.anodeAlignTableAxisX.source.posAbsolute,
                           intOut := "Unit1.Em4.HmiInterface".intCondition.Axis_15.Position.intOut);
   #_w1 := NOT (NOT #FALSE) AND "Unit1.Em4.ControlNodes".cm.Interlock.anodeAlignTableAxisX.source.posAbsolute[4];
   IF #_w1 THEN "Unit1.Em4.ControlNodes".cmAnodeAlignTableAxisX.commands.selectSetPosition := 4; END_IF;
   "Unit1.Em4.ControlNodes".cm.axisCommand.anodeAlignTableAxisX.posAbsolute[4] := #_w1;
END_REGION

REGION Network 175: CmAnodeAlignTableAxisX Position Absolute Position5
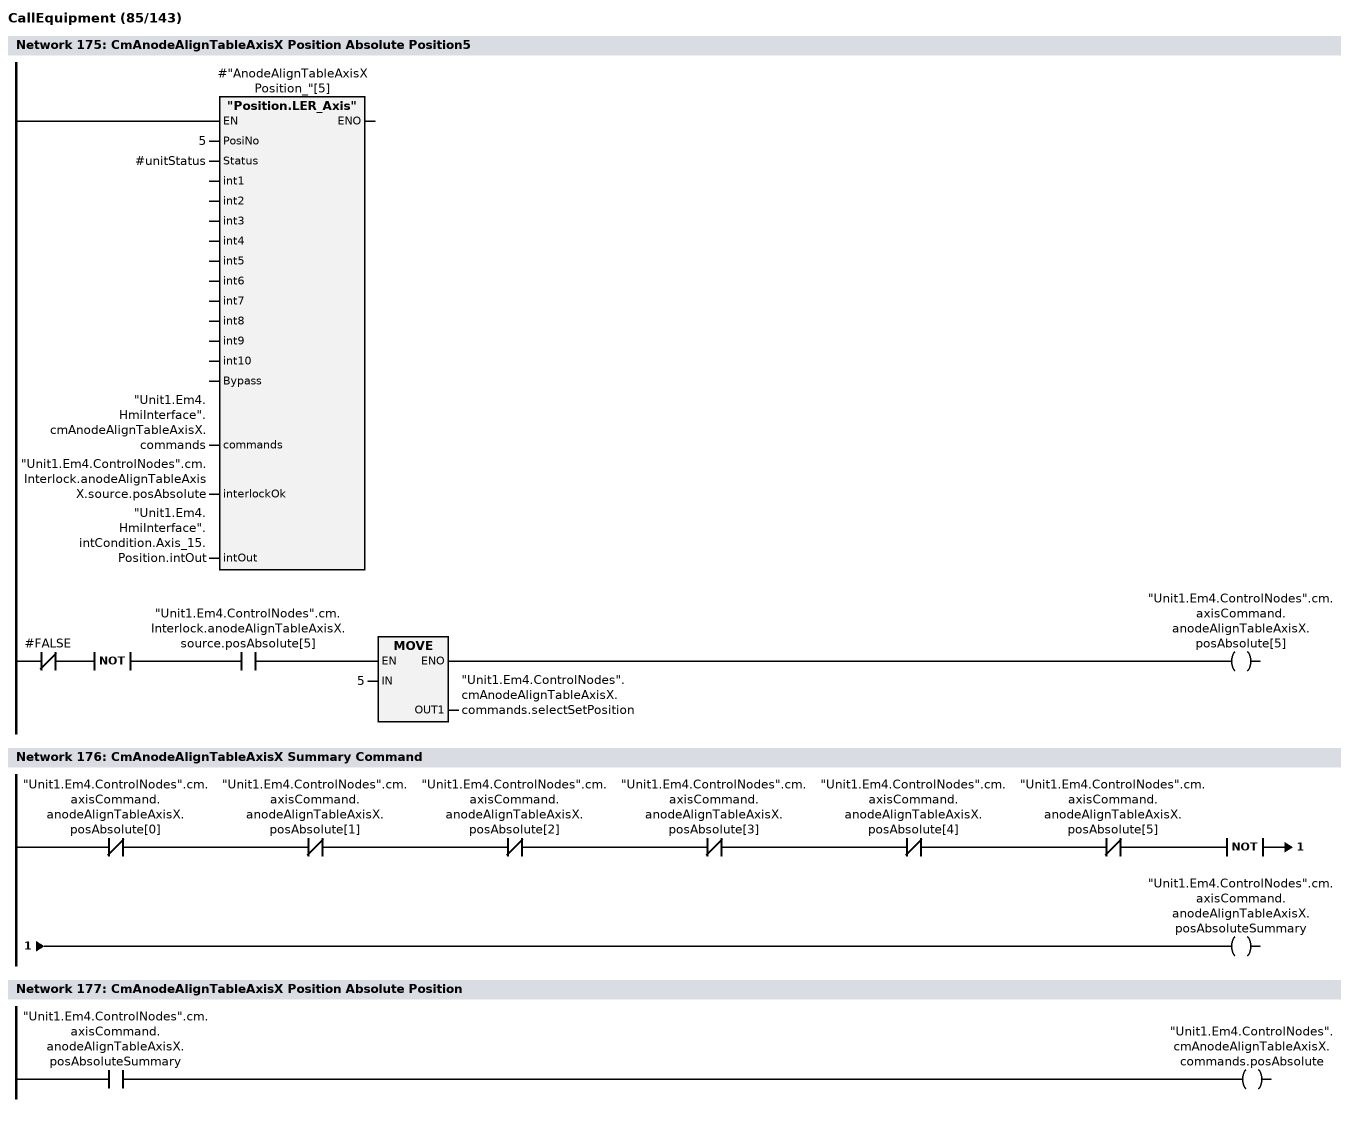
   RUNG wire#powerrail
      #"AnodeAlignTableAxisX Position_"[5](PosiNo := 5, Status := #unitStatus, int1 :=, int2 :=, int3 :=, int4 :=, int5 :=, int6 :=, int7 :=, int8 :=, int9 :=, int10 :=, Bypass :=, commands := "Unit1.Em4.HmiInterface".cmAnodeAlignTableAxisX.commands, interlockOk := "Unit1.Em4.ControlNodes".cm.Interlock.anodeAlignTableAxisX.source.posAbsolute, intOut := "Unit1.Em4.HmiInterface".intCondition.Axis_15.Position.intOut)
   END_RUNG
   RUNG wire#powerrail
      I_Contact( #FALSE )
      Not()
      Contact( "Unit1.Em4.ControlNodes".cm.Interlock.anodeAlignTableAxisX.source.posAbsolute[5] )
      Move(in := 5, out1 => "Unit1.Em4.ControlNodes".cmAnodeAlignTableAxisX.commands.selectSetPosition)
      Coil( "Unit1.Em4.ControlNodes".cm.axisCommand.anodeAlignTableAxisX.posAbsolute[5] )
   END_RUNG
   // the same network as SCL:
   #"AnodeAlignTableAxisX Position_"[5](PosiNo := 5,   // "Position.LER_Axis"
                           Status := #unitStatus,
                           commands := "Unit1.Em4.HmiInterface".cmAnodeAlignTableAxisX.commands,
                           interlockOk := "Unit1.Em4.ControlNodes".cm.Interlock.anodeAlignTableAxisX.source.posAbsolute,
                           intOut := "Unit1.Em4.HmiInterface".intCondition.Axis_15.Position.intOut);
   #_w1 := NOT (NOT #FALSE) AND "Unit1.Em4.ControlNodes".cm.Interlock.anodeAlignTableAxisX.source.posAbsolute[5];
   IF #_w1 THEN "Unit1.Em4.ControlNodes".cmAnodeAlignTableAxisX.commands.selectSetPosition := 5; END_IF;
   "Unit1.Em4.ControlNodes".cm.axisCommand.anodeAlignTableAxisX.posAbsolute[5] := #_w1;
END_REGION

REGION Network 176: CmAnodeAlignTableAxisX Summary Command
   RUNG wire#powerrail
      I_Contact( "Unit1.Em4.ControlNodes".cm.axisCommand.anodeAlignTableAxisX.posAbsolute[0] )
      I_Contact( "Unit1.Em4.ControlNodes".cm.axisCommand.anodeAlignTableAxisX.posAbsolute[1] )
      I_Contact( "Unit1.Em4.ControlNodes".cm.axisCommand.anodeAlignTableAxisX.posAbsolute[2] )
      I_Contact( "Unit1.Em4.ControlNodes".cm.axisCommand.anodeAlignTableAxisX.posAbsolute[3] )
      I_Contact( "Unit1.Em4.ControlNodes".cm.axisCommand.anodeAlignTableAxisX.posAbsolute[4] )
      I_Contact( "Unit1.Em4.ControlNodes".cm.axisCommand.anodeAlignTableAxisX.posAbsolute[5] )
      Not()
      Coil( "Unit1.Em4.ControlNodes".cm.axisCommand.anodeAlignTableAxisX.posAbsoluteSummary )
   END_RUNG
   // the same network as SCL:
   "Unit1.Em4.ControlNodes".cm.axisCommand.anodeAlignTableAxisX.posAbsoluteSummary := NOT (NOT "Unit1.Em4.ControlNodes".cm.axisCommand.anodeAlignTableAxisX.posAbsolute[0] AND NOT "Unit1.Em4.ControlNodes".cm.axisCommand.anodeAlignTableAxisX.posAbsolute[1] AND NOT "Unit1.Em4.ControlNodes".cm.axisCommand.anodeAlignTableAxisX.posAbsolute[2] AND NOT "Unit1.Em4.ControlNodes".cm.axisCommand.anodeAlignTableAxisX.posAbsolute[3] AND NOT "Unit1.Em4.ControlNodes".cm.axisCommand.anodeAlignTableAxisX.posAbsolute[4] AND NOT "Unit1.Em4.ControlNodes".cm.axisCommand.anodeAlignTableAxisX.posAbsolute[5]);
END_REGION

REGION Network 177: CmAnodeAlignTableAxisX Position Absolute Position
   RUNG wire#powerrail
      Contact( "Unit1.Em4.ControlNodes".cm.axisCommand.anodeAlignTableAxisX.posAbsoluteSummary )
      Coil( "Unit1.Em4.ControlNodes".cmAnodeAlignTableAxisX.commands.posAbsolute )
   END_RUNG
   // the same network as SCL:
   "Unit1.Em4.ControlNodes".cmAnodeAlignTableAxisX.commands.posAbsolute := "Unit1.Em4.ControlNodes".cm.axisCommand.anodeAlignTableAxisX.posAbsoluteSummary;
END_REGION

REGION Network 178: CmAnodeAlignTableAxisX Interlock Summary
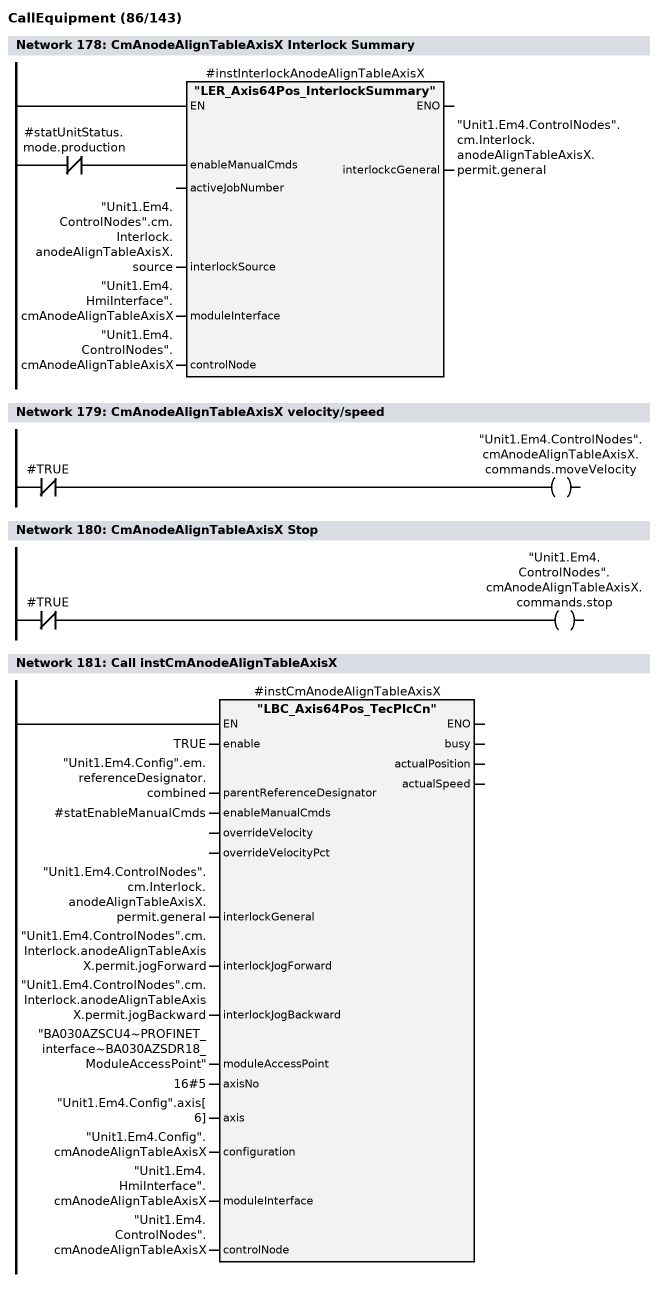
   RUNG wire#powerrail
      #instInterlockAnodeAlignTableAxisX(enableManualCmds := wire#w1, activeJobNumber :=, interlockSource := "Unit1.Em4.ControlNodes".cm.Interlock.anodeAlignTableAxisX.source, moduleInterface := "Unit1.Em4.HmiInterface".cmAnodeAlignTableAxisX, controlNode := "Unit1.Em4.ControlNodes".cmAnodeAlignTableAxisX, interlockcGeneral => "Unit1.Em4.ControlNodes".cm.Interlock.anodeAlignTableAxisX.permit.general)
   END_RUNG
   RUNG wire#powerrail
      I_Contact( #statUnitStatus.mode.production )
   END_RUNG wire#w1
   // the same network as SCL:
   #instInterlockAnodeAlignTableAxisX(enableManualCmds := NOT #statUnitStatus.mode.production,   // "LER_Axis64Pos_InterlockSummary"
                           interlockSource := "Unit1.Em4.ControlNodes".cm.Interlock.anodeAlignTableAxisX.source,
                           moduleInterface := "Unit1.Em4.HmiInterface".cmAnodeAlignTableAxisX,
                           controlNode := "Unit1.Em4.ControlNodes".cmAnodeAlignTableAxisX,
                           interlockcGeneral => "Unit1.Em4.ControlNodes".cm.Interlock.anodeAlignTableAxisX.permit.general);
END_REGION

REGION Network 179: CmAnodeAlignTableAxisX velocity/speed
   RUNG wire#powerrail
      I_Contact( #TRUE )
      Coil( "Unit1.Em4.ControlNodes".cmAnodeAlignTableAxisX.commands.moveVelocity )
   END_RUNG
   // the same network as SCL:
   "Unit1.Em4.ControlNodes".cmAnodeAlignTableAxisX.commands.moveVelocity := NOT #TRUE;
END_REGION

REGION Network 180: CmAnodeAlignTableAxisX Stop
   RUNG wire#powerrail
      I_Contact( #TRUE )
      Coil( "Unit1.Em4.ControlNodes".cmAnodeAlignTableAxisX.commands.stop )
   END_RUNG
   // the same network as SCL:
   "Unit1.Em4.ControlNodes".cmAnodeAlignTableAxisX.commands.stop := NOT #TRUE;
END_REGION

REGION Network 181: Call instCmAnodeAlignTableAxisX
   RUNG wire#powerrail
      #instCmAnodeAlignTableAxisX(enable := TRUE, parentReferenceDesignator := "Unit1.Em4.Config".em.referenceDesignator.combined, enableManualCmds := #statEnableManualCmds, overrideVelocity :=, overrideVelocityPct :=, interlockGeneral := "Unit1.Em4.ControlNodes".cm.Interlock.anodeAlignTableAxisX.permit.general, interlockJogForward := "Unit1.Em4.ControlNodes".cm.Interlock.anodeAlignTableAxisX.permit.jogForward, interlockJogBackward := "Unit1.Em4.ControlNodes".cm.Interlock.anodeAlignTableAxisX.permit.jogBackward, moduleAccessPoint := "BA030AZSCU4~PROFINET_interface~BA030AZSDR18_ModuleAccessPoint", axisNo := 16#5, axis := "Unit1.Em4.Config".axis[6], configuration := "Unit1.Em4.Config".cmAnodeAlignTableAxisX, moduleInterface := "Unit1.Em4.HmiInterface".cmAnodeAlignTableAxisX, controlNode := "Unit1.Em4.ControlNodes".cmAnodeAlignTableAxisX, busy =>, actualPosition =>, actualSpeed =>)
   END_RUNG
   // the same network as SCL:
   #instCmAnodeAlignTableAxisX(enable := TRUE,   // "LBC_Axis64Pos_TecPlcCn"
                           parentReferenceDesignator := "Unit1.Em4.Config".em.referenceDesignator.combined,
                           enableManualCmds := #statEnableManualCmds,
                           interlockGeneral := "Unit1.Em4.ControlNodes".cm.Interlock.anodeAlignTableAxisX.permit.general,
                           interlockJogForward := "Unit1.Em4.ControlNodes".cm.Interlock.anodeAlignTableAxisX.permit.jogForward,
                           interlockJogBackward := "Unit1.Em4.ControlNodes".cm.Interlock.anodeAlignTableAxisX.permit.jogBackward,
                           moduleAccessPoint := "BA030AZSCU4~PROFINET_interface~BA030AZSDR18_ModuleAccessPoint",
                           axisNo := 16#5,
                           axis := "Unit1.Em4.Config".axis[6],
                           configuration := "Unit1.Em4.Config".cmAnodeAlignTableAxisX,
                           moduleInterface := "Unit1.Em4.HmiInterface".cmAnodeAlignTableAxisX,
                           controlNode := "Unit1.Em4.ControlNodes".cmAnodeAlignTableAxisX);
END_REGION

REGION Network 182: CmAnodeAlignTableAxisX SoftCam
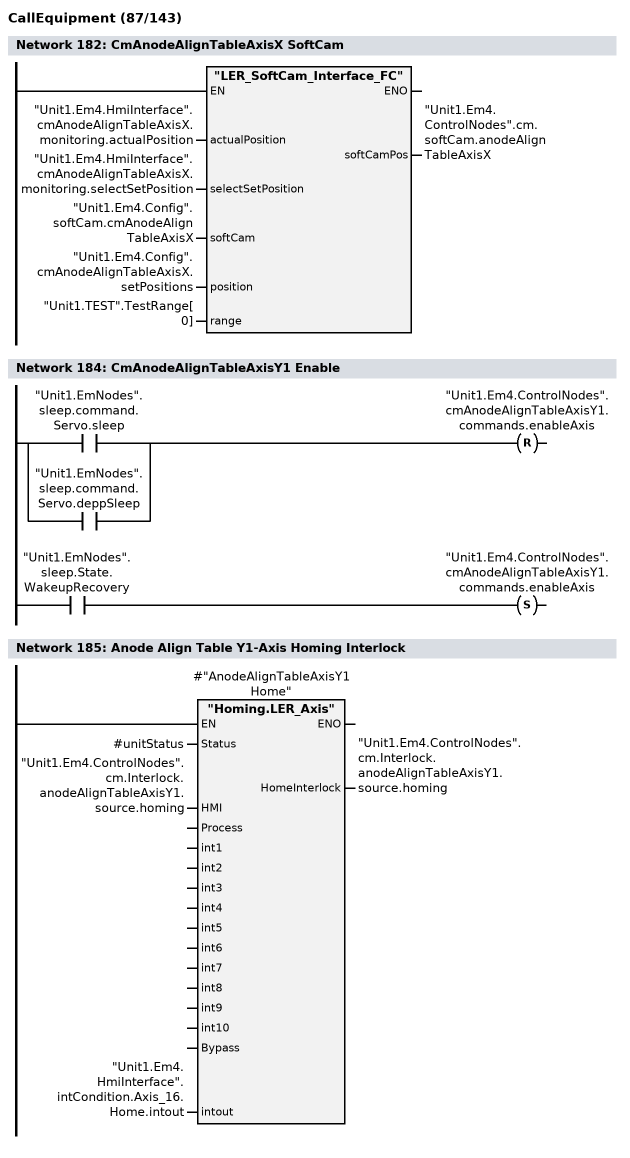
   RUNG wire#powerrail
      "LER_SoftCam_Interface_FC"(actualPosition := "Unit1.Em4.HmiInterface".cmAnodeAlignTableAxisX.monitoring.actualPosition, selectSetPosition := "Unit1.Em4.HmiInterface".cmAnodeAlignTableAxisX.monitoring.selectSetPosition, softCam := "Unit1.Em4.Config".softCam.cmAnodeAlignTableAxisX, position := "Unit1.Em4.Config".cmAnodeAlignTableAxisX.setPositions, range := "Unit1.TEST".TestRange[0], softCamPos => "Unit1.Em4.ControlNodes".cm.softCam.anodeAlignTableAxisX)
   END_RUNG
   // the same network as SCL:
   "LER_SoftCam_Interface_FC"(actualPosition := "Unit1.Em4.HmiInterface".cmAnodeAlignTableAxisX.monitoring.actualPosition,
                           selectSetPosition := "Unit1.Em4.HmiInterface".cmAnodeAlignTableAxisX.monitoring.selectSetPosition,
                           softCam := "Unit1.Em4.Config".softCam.cmAnodeAlignTableAxisX,
                           position := "Unit1.Em4.Config".cmAnodeAlignTableAxisX.setPositions,
                           range := "Unit1.TEST".TestRange[0],
                           softCamPos => "Unit1.Em4.ControlNodes".cm.softCam.anodeAlignTableAxisX);
END_REGION

REGION Network 184: CmAnodeAlignTableAxisY1 Enable
   RUNG wire#powerrail
      Contact( "Unit1.EmNodes".sleep.command.Servo.sleep )
      wire#w1
      R_Coil( "Unit1.Em4.ControlNodes".cmAnodeAlignTableAxisY1.commands.enableAxis )
   END_RUNG
   RUNG wire#powerrail
      Contact( "Unit1.EmNodes".sleep.command.Servo.deppSleep )
   END_RUNG wire#w1
   RUNG wire#powerrail
      Contact( "Unit1.EmNodes".sleep.State.WakeupRecovery )
      S_Coil( "Unit1.Em4.ControlNodes".cmAnodeAlignTableAxisY1.commands.enableAxis )
   END_RUNG
   // the same network as SCL:
   IF "Unit1.EmNodes".sleep.command.Servo.sleep OR "Unit1.EmNodes".sleep.command.Servo.deppSleep THEN
       "Unit1.Em4.ControlNodes".cmAnodeAlignTableAxisY1.commands.enableAxis := FALSE;
   END_IF;
   IF "Unit1.EmNodes".sleep.State.WakeupRecovery THEN
       "Unit1.Em4.ControlNodes".cmAnodeAlignTableAxisY1.commands.enableAxis := TRUE;
   END_IF;
END_REGION

REGION Network 185: Anode Align Table Y1-Axis Homing Interlock
   RUNG wire#powerrail
      #"AnodeAlignTableAxisY1 Home"(Status := #unitStatus, HMI := "Unit1.Em4.ControlNodes".cm.Interlock.anodeAlignTableAxisY1.source.homing, Process :=, int1 :=, int2 :=, int3 :=, int4 :=, int5 :=, int6 :=, int7 :=, int8 :=, int9 :=, int10 :=, Bypass :=, intout := "Unit1.Em4.HmiInterface".intCondition.Axis_16.Home.intout, HomeInterlock => "Unit1.Em4.ControlNodes".cm.Interlock.anodeAlignTableAxisY1.source.homing)
   END_RUNG
   // the same network as SCL:
   #"AnodeAlignTableAxisY1 Home"(Status := #unitStatus,   // "Homing.LER_Axis"
                           HMI := "Unit1.Em4.ControlNodes".cm.Interlock.anodeAlignTableAxisY1.source.homing,
                           intout := "Unit1.Em4.HmiInterface".intCondition.Axis_16.Home.intout,
                           HomeInterlock => "Unit1.Em4.ControlNodes".cm.Interlock.anodeAlignTableAxisY1.source.homing);
END_REGION

REGION Network 186: CmAnodeAlignTableAxisY1 Position Absolute Jog
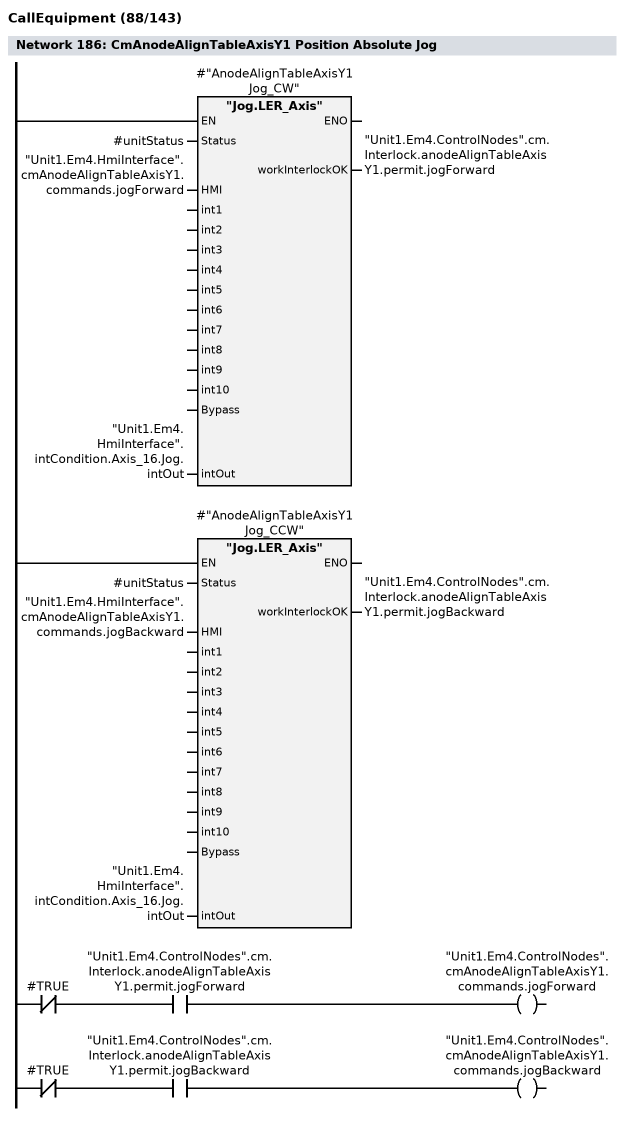
   RUNG wire#powerrail
      #"AnodeAlignTableAxisY1 Jog_CW"(Status := #unitStatus, HMI := "Unit1.Em4.HmiInterface".cmAnodeAlignTableAxisY1.commands.jogForward, int1 :=, int2 :=, int3 :=, int4 :=, int5 :=, int6 :=, int7 :=, int8 :=, int9 :=, int10 :=, Bypass :=, intOut := "Unit1.Em4.HmiInterface".intCondition.Axis_16.Jog.intOut, workInterlockOK => "Unit1.Em4.ControlNodes".cm.Interlock.anodeAlignTableAxisY1.permit.jogForward)
   END_RUNG
   RUNG wire#powerrail
      #"AnodeAlignTableAxisY1 Jog_CCW"(Status := #unitStatus, HMI := "Unit1.Em4.HmiInterface".cmAnodeAlignTableAxisY1.commands.jogBackward, int1 :=, int2 :=, int3 :=, int4 :=, int5 :=, int6 :=, int7 :=, int8 :=, int9 :=, int10 :=, Bypass :=, intOut := "Unit1.Em4.HmiInterface".intCondition.Axis_16.Jog.intOut, workInterlockOK => "Unit1.Em4.ControlNodes".cm.Interlock.anodeAlignTableAxisY1.permit.jogBackward)
   END_RUNG
   RUNG wire#powerrail
      I_Contact( #TRUE )
      Contact( "Unit1.Em4.ControlNodes".cm.Interlock.anodeAlignTableAxisY1.permit.jogForward )
      Coil( "Unit1.Em4.ControlNodes".cmAnodeAlignTableAxisY1.commands.jogForward )
   END_RUNG
   RUNG wire#powerrail
      I_Contact( #TRUE )
      Contact( "Unit1.Em4.ControlNodes".cm.Interlock.anodeAlignTableAxisY1.permit.jogBackward )
      Coil( "Unit1.Em4.ControlNodes".cmAnodeAlignTableAxisY1.commands.jogBackward )
   END_RUNG
   // the same network as SCL:
   #"AnodeAlignTableAxisY1 Jog_CW"(Status := #unitStatus,   // "Jog.LER_Axis"
                           HMI := "Unit1.Em4.HmiInterface".cmAnodeAlignTableAxisY1.commands.jogForward,
                           intOut := "Unit1.Em4.HmiInterface".intCondition.Axis_16.Jog.intOut,
                           workInterlockOK => "Unit1.Em4.ControlNodes".cm.Interlock.anodeAlignTableAxisY1.permit.jogForward);
   #"AnodeAlignTableAxisY1 Jog_CCW"(Status := #unitStatus,   // "Jog.LER_Axis"
                           HMI := "Unit1.Em4.HmiInterface".cmAnodeAlignTableAxisY1.commands.jogBackward,
                           intOut := "Unit1.Em4.HmiInterface".intCondition.Axis_16.Jog.intOut,
                           workInterlockOK => "Unit1.Em4.ControlNodes".cm.Interlock.anodeAlignTableAxisY1.permit.jogBackward);
   "Unit1.Em4.ControlNodes".cmAnodeAlignTableAxisY1.commands.jogForward := NOT #TRUE AND "Unit1.Em4.ControlNodes".cm.Interlock.anodeAlignTableAxisY1.permit.jogForward;
   "Unit1.Em4.ControlNodes".cmAnodeAlignTableAxisY1.commands.jogBackward := NOT #TRUE AND "Unit1.Em4.ControlNodes".cm.Interlock.anodeAlignTableAxisY1.permit.jogBackward;
END_REGION

REGION Network 187: CmAnodeAlignTableAxisY1 Position Absolute Position0
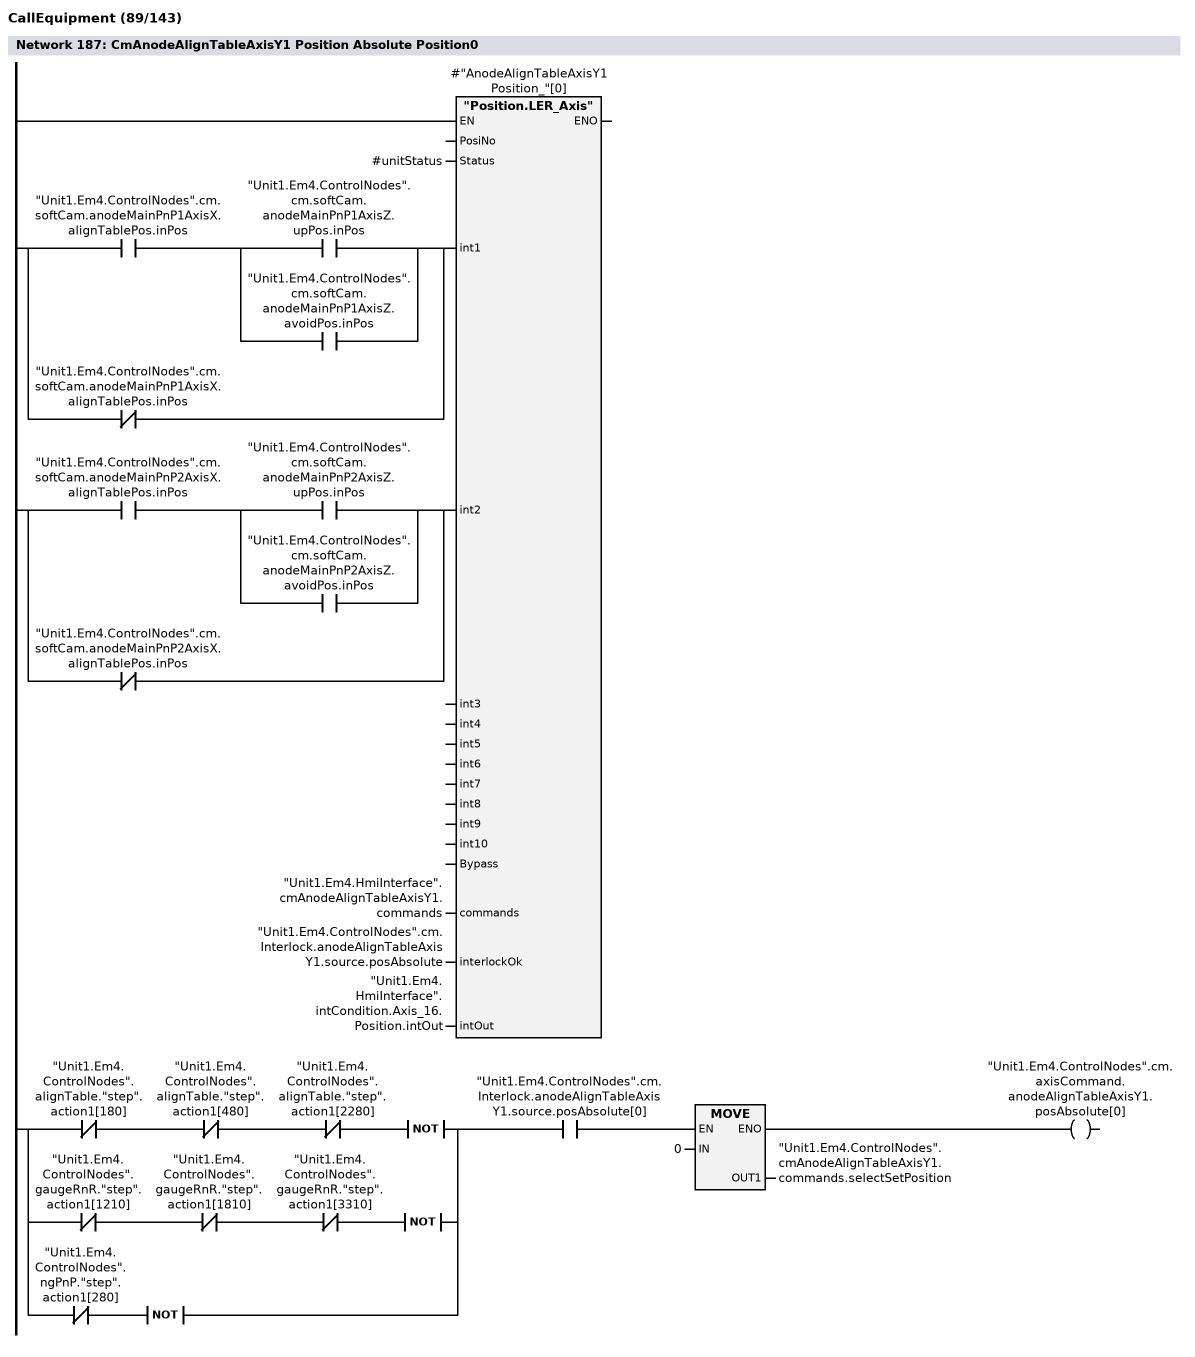
   RUNG wire#powerrail
      #"AnodeAlignTableAxisY1 Position_"[0](int1 := wire#w2, int2 := wire#w4, PosiNo :=, Status := #unitStatus, int3 :=, int4 :=, int5 :=, int6 :=, int7 :=, int8 :=, int9 :=, int10 :=, Bypass :=, commands := "Unit1.Em4.HmiInterface".cmAnodeAlignTableAxisY1.commands, interlockOk := "Unit1.Em4.ControlNodes".cm.Interlock.anodeAlignTableAxisY1.source.posAbsolute, intOut := "Unit1.Em4.HmiInterface".intCondition.Axis_16.Position.intOut)
   END_RUNG
   RUNG wire#powerrail
      Contact( "Unit1.Em4.ControlNodes".cm.softCam.anodeMainPnP1AxisX.alignTablePos.inPos )
      wire#w1
      Contact( "Unit1.Em4.ControlNodes".cm.softCam.anodeMainPnP1AxisZ.upPos.inPos )
   END_RUNG wire#w2
   RUNG wire#w1
      Contact( "Unit1.Em4.ControlNodes".cm.softCam.anodeMainPnP1AxisZ.avoidPos.inPos )
   END_RUNG wire#w2
   RUNG wire#powerrail
      I_Contact( "Unit1.Em4.ControlNodes".cm.softCam.anodeMainPnP1AxisX.alignTablePos.inPos )
   END_RUNG wire#w2
   RUNG wire#powerrail
      Contact( "Unit1.Em4.ControlNodes".cm.softCam.anodeMainPnP2AxisX.alignTablePos.inPos )
      wire#w3
      Contact( "Unit1.Em4.ControlNodes".cm.softCam.anodeMainPnP2AxisZ.upPos.inPos )
   END_RUNG wire#w4
   RUNG wire#w3
      Contact( "Unit1.Em4.ControlNodes".cm.softCam.anodeMainPnP2AxisZ.avoidPos.inPos )
   END_RUNG wire#w4
   RUNG wire#powerrail
      I_Contact( "Unit1.Em4.ControlNodes".cm.softCam.anodeMainPnP2AxisX.alignTablePos.inPos )
   END_RUNG wire#w4
   RUNG wire#powerrail
      I_Contact( "Unit1.Em4.ControlNodes".alignTable."step".action1[180] )
      I_Contact( "Unit1.Em4.ControlNodes".alignTable."step".action1[480] )
      I_Contact( "Unit1.Em4.ControlNodes".alignTable."step".action1[2280] )
      Not()
      wire#w5
      Contact( "Unit1.Em4.ControlNodes".cm.Interlock.anodeAlignTableAxisY1.source.posAbsolute[0] )
      Move(in := 0, out1 => "Unit1.Em4.ControlNodes".cmAnodeAlignTableAxisY1.commands.selectSetPosition)
      Coil( "Unit1.Em4.ControlNodes".cm.axisCommand.anodeAlignTableAxisY1.posAbsolute[0] )
   END_RUNG
   RUNG wire#powerrail
      I_Contact( "Unit1.Em4.ControlNodes".gaugeRnR."step".action1[1210] )
      I_Contact( "Unit1.Em4.ControlNodes".gaugeRnR."step".action1[1810] )
      I_Contact( "Unit1.Em4.ControlNodes".gaugeRnR."step".action1[3310] )
      Not()
   END_RUNG wire#w5
   RUNG wire#powerrail
      I_Contact( "Unit1.Em4.ControlNodes".ngPnP."step".action1[280] )
      Not()
   END_RUNG wire#w5
   // the same network as SCL:
   #"AnodeAlignTableAxisY1 Position_"[0](Status := #unitStatus,   // "Position.LER_Axis"
                           int1 := ("Unit1.Em4.ControlNodes".cm.softCam.anodeMainPnP1AxisX.alignTablePos.inPos AND ("Unit1.Em4.ControlNodes".cm.softCam.anodeMainPnP1AxisZ.upPos.inPos OR "Unit1.Em4.ControlNodes".cm.softCam.anodeMainPnP1AxisZ.avoidPos.inPos)) OR NOT "Unit1.Em4.ControlNodes".cm.softCam.anodeMainPnP1AxisX.alignTablePos.inPos,
                           int2 := ("Unit1.Em4.ControlNodes".cm.softCam.anodeMainPnP2AxisX.alignTablePos.inPos AND ("Unit1.Em4.ControlNodes".cm.softCam.anodeMainPnP2AxisZ.upPos.inPos OR "Unit1.Em4.ControlNodes".cm.softCam.anodeMainPnP2AxisZ.avoidPos.inPos)) OR NOT "Unit1.Em4.ControlNodes".cm.softCam.anodeMainPnP2AxisX.alignTablePos.inPos,
                           commands := "Unit1.Em4.HmiInterface".cmAnodeAlignTableAxisY1.commands,
                           interlockOk := "Unit1.Em4.ControlNodes".cm.Interlock.anodeAlignTableAxisY1.source.posAbsolute,
                           intOut := "Unit1.Em4.HmiInterface".intCondition.Axis_16.Position.intOut);
   #_w1 := (NOT (NOT "Unit1.Em4.ControlNodes".alignTable."step".action1[180] AND NOT "Unit1.Em4.ControlNodes".alignTable."step".action1[480] AND NOT "Unit1.Em4.ControlNodes".alignTable."step".action1[2280]) OR NOT (NOT "Unit1.Em4.ControlNodes".gaugeRnR."step".action1[1210] AND NOT "Unit1.Em4.ControlNodes".gaugeRnR."step".action1[1810] AND NOT "Unit1.Em4.ControlNodes".gaugeRnR."step".action1[3310]) OR NOT (NOT "Unit1.Em4.ControlNodes".ngPnP."step".action1[280])) AND "Unit1.Em4.ControlNodes".cm.Interlock.anodeAlignTableAxisY1.source.posAbsolute[0];
   IF #_w1 THEN "Unit1.Em4.ControlNodes".cmAnodeAlignTableAxisY1.commands.selectSetPosition := 0; END_IF;
   "Unit1.Em4.ControlNodes".cm.axisCommand.anodeAlignTableAxisY1.posAbsolute[0] := #_w1;
END_REGION

REGION Network 188: CmAnodeAlignTableAxisY1 Position Absolute Position1
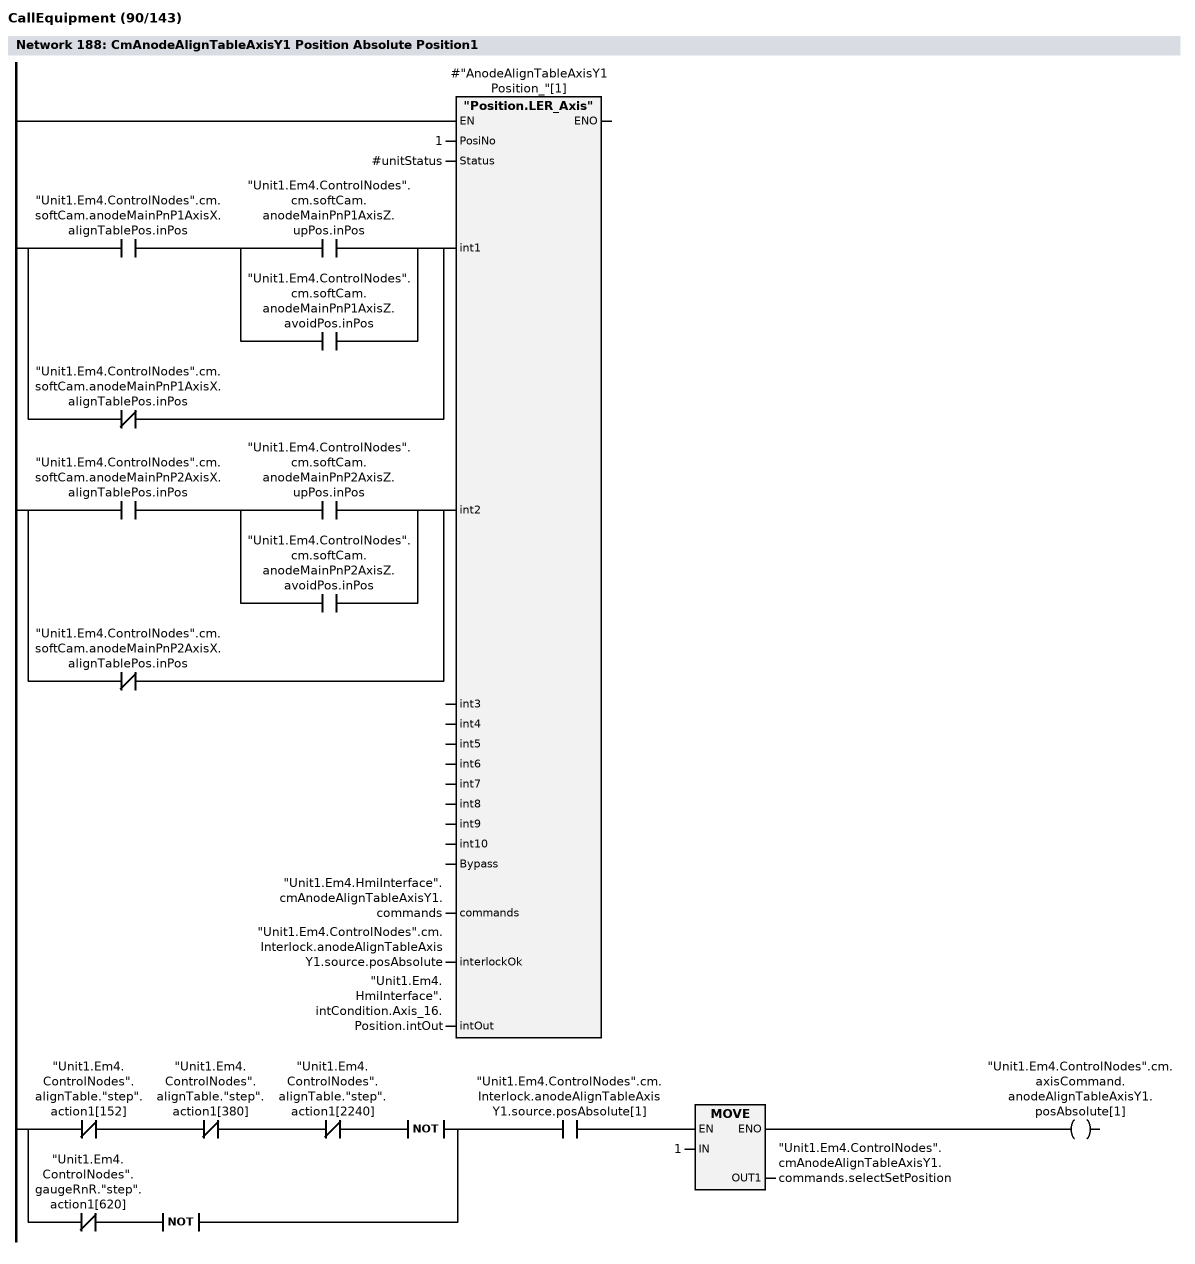
   RUNG wire#powerrail
      #"AnodeAlignTableAxisY1 Position_"[1](int1 := wire#w2, int2 := wire#w4, PosiNo := 1, Status := #unitStatus, int3 :=, int4 :=, int5 :=, int6 :=, int7 :=, int8 :=, int9 :=, int10 :=, Bypass :=, commands := "Unit1.Em4.HmiInterface".cmAnodeAlignTableAxisY1.commands, interlockOk := "Unit1.Em4.ControlNodes".cm.Interlock.anodeAlignTableAxisY1.source.posAbsolute, intOut := "Unit1.Em4.HmiInterface".intCondition.Axis_16.Position.intOut)
   END_RUNG
   RUNG wire#powerrail
      Contact( "Unit1.Em4.ControlNodes".cm.softCam.anodeMainPnP1AxisX.alignTablePos.inPos )
      wire#w1
      Contact( "Unit1.Em4.ControlNodes".cm.softCam.anodeMainPnP1AxisZ.upPos.inPos )
   END_RUNG wire#w2
   RUNG wire#w1
      Contact( "Unit1.Em4.ControlNodes".cm.softCam.anodeMainPnP1AxisZ.avoidPos.inPos )
   END_RUNG wire#w2
   RUNG wire#powerrail
      I_Contact( "Unit1.Em4.ControlNodes".cm.softCam.anodeMainPnP1AxisX.alignTablePos.inPos )
   END_RUNG wire#w2
   RUNG wire#powerrail
      Contact( "Unit1.Em4.ControlNodes".cm.softCam.anodeMainPnP2AxisX.alignTablePos.inPos )
      wire#w3
      Contact( "Unit1.Em4.ControlNodes".cm.softCam.anodeMainPnP2AxisZ.upPos.inPos )
   END_RUNG wire#w4
   RUNG wire#w3
      Contact( "Unit1.Em4.ControlNodes".cm.softCam.anodeMainPnP2AxisZ.avoidPos.inPos )
   END_RUNG wire#w4
   RUNG wire#powerrail
      I_Contact( "Unit1.Em4.ControlNodes".cm.softCam.anodeMainPnP2AxisX.alignTablePos.inPos )
   END_RUNG wire#w4
   RUNG wire#powerrail
      I_Contact( "Unit1.Em4.ControlNodes".alignTable."step".action1[152] )
      I_Contact( "Unit1.Em4.ControlNodes".alignTable."step".action1[380] )
      I_Contact( "Unit1.Em4.ControlNodes".alignTable."step".action1[2240] )
      Not()
      wire#w5
      Contact( "Unit1.Em4.ControlNodes".cm.Interlock.anodeAlignTableAxisY1.source.posAbsolute[1] )
      Move(in := 1, out1 => "Unit1.Em4.ControlNodes".cmAnodeAlignTableAxisY1.commands.selectSetPosition)
      Coil( "Unit1.Em4.ControlNodes".cm.axisCommand.anodeAlignTableAxisY1.posAbsolute[1] )
   END_RUNG
   RUNG wire#powerrail
      I_Contact( "Unit1.Em4.ControlNodes".gaugeRnR."step".action1[620] )
      Not()
   END_RUNG wire#w5
   // the same network as SCL:
   #"AnodeAlignTableAxisY1 Position_"[1](PosiNo := 1,   // "Position.LER_Axis"
                           Status := #unitStatus,
                           int1 := ("Unit1.Em4.ControlNodes".cm.softCam.anodeMainPnP1AxisX.alignTablePos.inPos AND ("Unit1.Em4.ControlNodes".cm.softCam.anodeMainPnP1AxisZ.upPos.inPos OR "Unit1.Em4.ControlNodes".cm.softCam.anodeMainPnP1AxisZ.avoidPos.inPos)) OR NOT "Unit1.Em4.ControlNodes".cm.softCam.anodeMainPnP1AxisX.alignTablePos.inPos,
                           int2 := ("Unit1.Em4.ControlNodes".cm.softCam.anodeMainPnP2AxisX.alignTablePos.inPos AND ("Unit1.Em4.ControlNodes".cm.softCam.anodeMainPnP2AxisZ.upPos.inPos OR "Unit1.Em4.ControlNodes".cm.softCam.anodeMainPnP2AxisZ.avoidPos.inPos)) OR NOT "Unit1.Em4.ControlNodes".cm.softCam.anodeMainPnP2AxisX.alignTablePos.inPos,
                           commands := "Unit1.Em4.HmiInterface".cmAnodeAlignTableAxisY1.commands,
                           interlockOk := "Unit1.Em4.ControlNodes".cm.Interlock.anodeAlignTableAxisY1.source.posAbsolute,
                           intOut := "Unit1.Em4.HmiInterface".intCondition.Axis_16.Position.intOut);
   #_w1 := (NOT (NOT "Unit1.Em4.ControlNodes".alignTable."step".action1[152] AND NOT "Unit1.Em4.ControlNodes".alignTable."step".action1[380] AND NOT "Unit1.Em4.ControlNodes".alignTable."step".action1[2240]) OR NOT (NOT "Unit1.Em4.ControlNodes".gaugeRnR."step".action1[620])) AND "Unit1.Em4.ControlNodes".cm.Interlock.anodeAlignTableAxisY1.source.posAbsolute[1];
   IF #_w1 THEN "Unit1.Em4.ControlNodes".cmAnodeAlignTableAxisY1.commands.selectSetPosition := 1; END_IF;
   "Unit1.Em4.ControlNodes".cm.axisCommand.anodeAlignTableAxisY1.posAbsolute[1] := #_w1;
END_REGION

REGION Network 189: CmAnodeAlignTableAxisY1 Position Absolute Position2
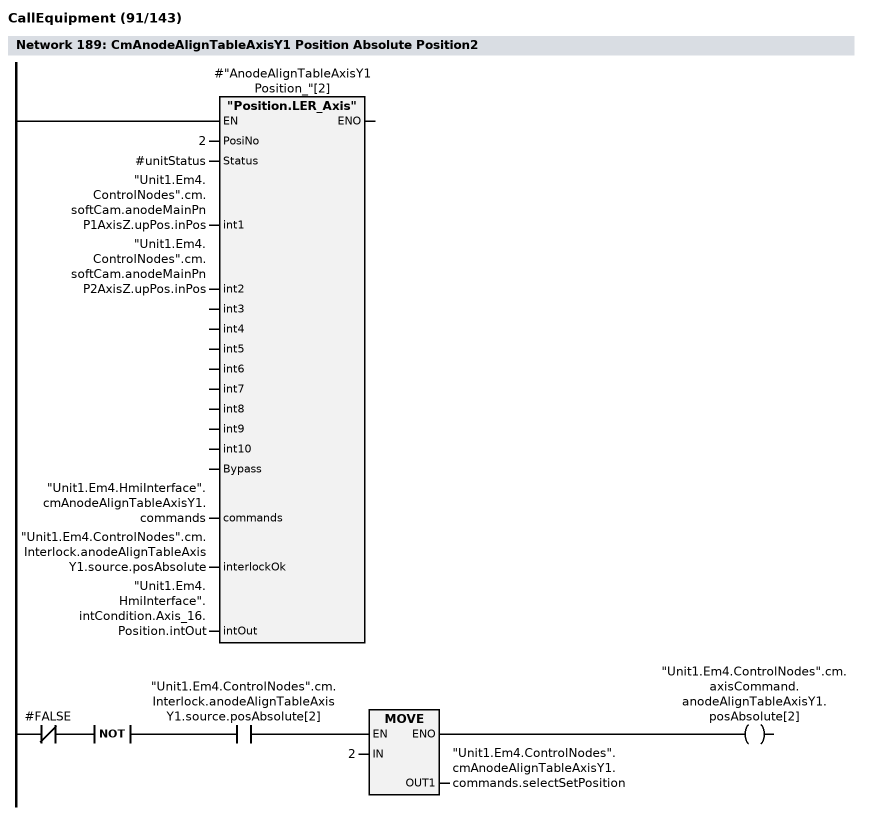
   RUNG wire#powerrail
      #"AnodeAlignTableAxisY1 Position_"[2](PosiNo := 2, Status := #unitStatus, int1 := "Unit1.Em4.ControlNodes".cm.softCam.anodeMainPnP1AxisZ.upPos.inPos, int2 := "Unit1.Em4.ControlNodes".cm.softCam.anodeMainPnP2AxisZ.upPos.inPos, int3 :=, int4 :=, int5 :=, int6 :=, int7 :=, int8 :=, int9 :=, int10 :=, Bypass :=, commands := "Unit1.Em4.HmiInterface".cmAnodeAlignTableAxisY1.commands, interlockOk := "Unit1.Em4.ControlNodes".cm.Interlock.anodeAlignTableAxisY1.source.posAbsolute, intOut := "Unit1.Em4.HmiInterface".intCondition.Axis_16.Position.intOut)
   END_RUNG
   RUNG wire#powerrail
      I_Contact( #FALSE )
      Not()
      Contact( "Unit1.Em4.ControlNodes".cm.Interlock.anodeAlignTableAxisY1.source.posAbsolute[2] )
      Move(in := 2, out1 => "Unit1.Em4.ControlNodes".cmAnodeAlignTableAxisY1.commands.selectSetPosition)
      Coil( "Unit1.Em4.ControlNodes".cm.axisCommand.anodeAlignTableAxisY1.posAbsolute[2] )
   END_RUNG
   // the same network as SCL:
   #"AnodeAlignTableAxisY1 Position_"[2](PosiNo := 2,   // "Position.LER_Axis"
                           Status := #unitStatus,
                           int1 := "Unit1.Em4.ControlNodes".cm.softCam.anodeMainPnP1AxisZ.upPos.inPos,
                           int2 := "Unit1.Em4.ControlNodes".cm.softCam.anodeMainPnP2AxisZ.upPos.inPos,
                           commands := "Unit1.Em4.HmiInterface".cmAnodeAlignTableAxisY1.commands,
                           interlockOk := "Unit1.Em4.ControlNodes".cm.Interlock.anodeAlignTableAxisY1.source.posAbsolute,
                           intOut := "Unit1.Em4.HmiInterface".intCondition.Axis_16.Position.intOut);
   #_w1 := NOT (NOT #FALSE) AND "Unit1.Em4.ControlNodes".cm.Interlock.anodeAlignTableAxisY1.source.posAbsolute[2];
   IF #_w1 THEN "Unit1.Em4.ControlNodes".cmAnodeAlignTableAxisY1.commands.selectSetPosition := 2; END_IF;
   "Unit1.Em4.ControlNodes".cm.axisCommand.anodeAlignTableAxisY1.posAbsolute[2] := #_w1;
END_REGION

REGION Network 190: CmAnodeAlignTableAxisY1 Position Absolute Position3
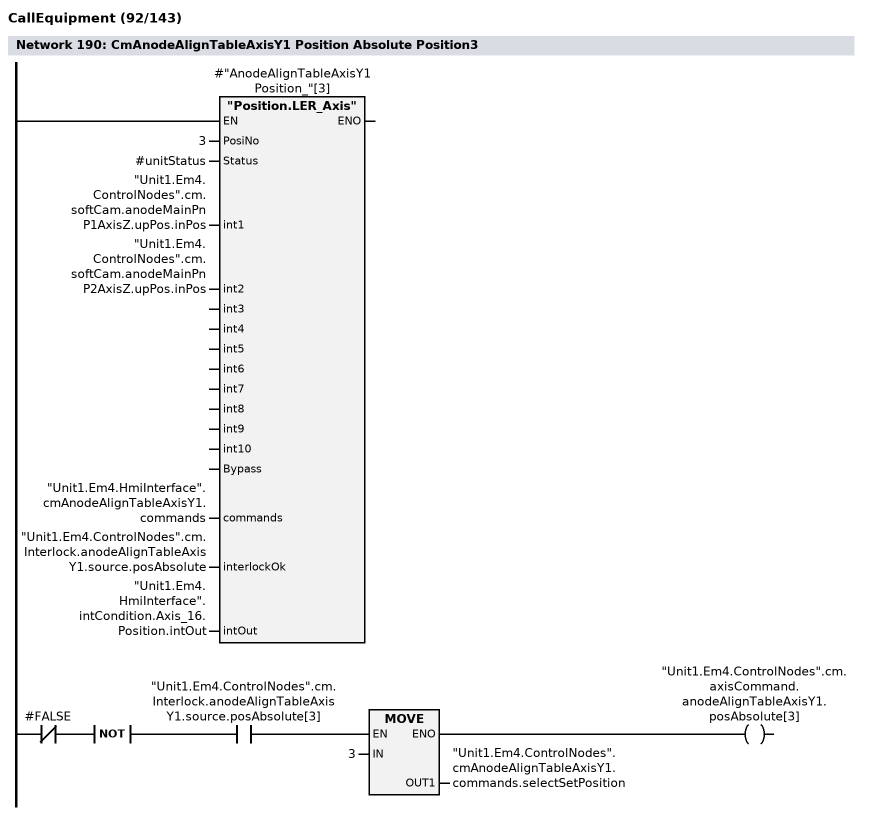
   RUNG wire#powerrail
      #"AnodeAlignTableAxisY1 Position_"[3](PosiNo := 3, Status := #unitStatus, int1 := "Unit1.Em4.ControlNodes".cm.softCam.anodeMainPnP1AxisZ.upPos.inPos, int2 := "Unit1.Em4.ControlNodes".cm.softCam.anodeMainPnP2AxisZ.upPos.inPos, int3 :=, int4 :=, int5 :=, int6 :=, int7 :=, int8 :=, int9 :=, int10 :=, Bypass :=, commands := "Unit1.Em4.HmiInterface".cmAnodeAlignTableAxisY1.commands, interlockOk := "Unit1.Em4.ControlNodes".cm.Interlock.anodeAlignTableAxisY1.source.posAbsolute, intOut := "Unit1.Em4.HmiInterface".intCondition.Axis_16.Position.intOut)
   END_RUNG
   RUNG wire#powerrail
      I_Contact( #FALSE )
      Not()
      Contact( "Unit1.Em4.ControlNodes".cm.Interlock.anodeAlignTableAxisY1.source.posAbsolute[3] )
      Move(in := 3, out1 => "Unit1.Em4.ControlNodes".cmAnodeAlignTableAxisY1.commands.selectSetPosition)
      Coil( "Unit1.Em4.ControlNodes".cm.axisCommand.anodeAlignTableAxisY1.posAbsolute[3] )
   END_RUNG
   // the same network as SCL:
   #"AnodeAlignTableAxisY1 Position_"[3](PosiNo := 3,   // "Position.LER_Axis"
                           Status := #unitStatus,
                           int1 := "Unit1.Em4.ControlNodes".cm.softCam.anodeMainPnP1AxisZ.upPos.inPos,
                           int2 := "Unit1.Em4.ControlNodes".cm.softCam.anodeMainPnP2AxisZ.upPos.inPos,
                           commands := "Unit1.Em4.HmiInterface".cmAnodeAlignTableAxisY1.commands,
                           interlockOk := "Unit1.Em4.ControlNodes".cm.Interlock.anodeAlignTableAxisY1.source.posAbsolute,
                           intOut := "Unit1.Em4.HmiInterface".intCondition.Axis_16.Position.intOut);
   #_w1 := NOT (NOT #FALSE) AND "Unit1.Em4.ControlNodes".cm.Interlock.anodeAlignTableAxisY1.source.posAbsolute[3];
   IF #_w1 THEN "Unit1.Em4.ControlNodes".cmAnodeAlignTableAxisY1.commands.selectSetPosition := 3; END_IF;
   "Unit1.Em4.ControlNodes".cm.axisCommand.anodeAlignTableAxisY1.posAbsolute[3] := #_w1;
END_REGION

REGION Network 191: CmAnodeAlignTableAxisY1 Position Absolute Position4
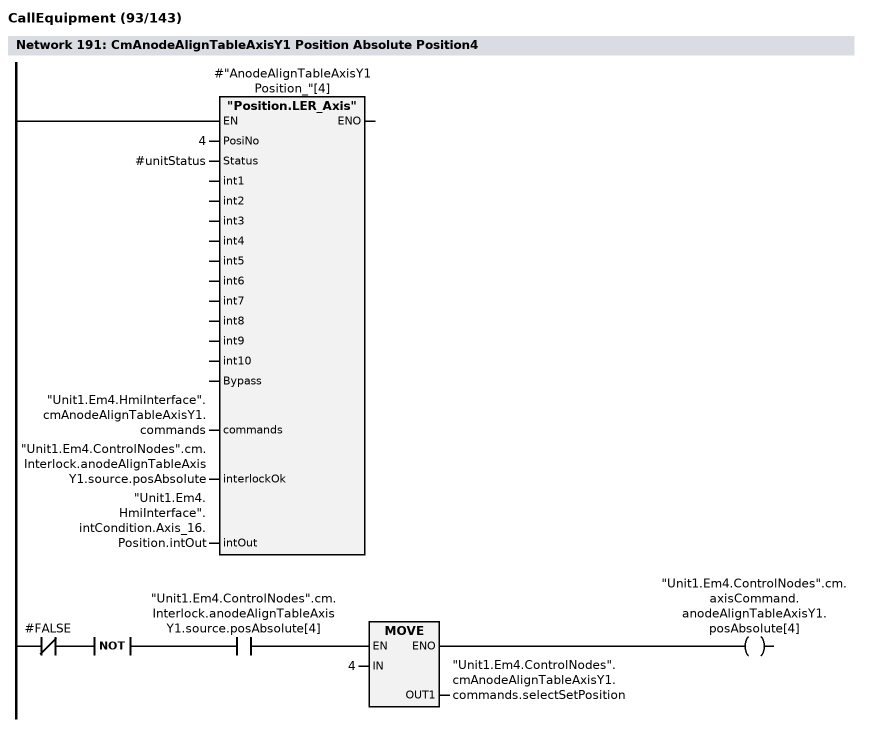
   RUNG wire#powerrail
      #"AnodeAlignTableAxisY1 Position_"[4](PosiNo := 4, Status := #unitStatus, int1 :=, int2 :=, int3 :=, int4 :=, int5 :=, int6 :=, int7 :=, int8 :=, int9 :=, int10 :=, Bypass :=, commands := "Unit1.Em4.HmiInterface".cmAnodeAlignTableAxisY1.commands, interlockOk := "Unit1.Em4.ControlNodes".cm.Interlock.anodeAlignTableAxisY1.source.posAbsolute, intOut := "Unit1.Em4.HmiInterface".intCondition.Axis_16.Position.intOut)
   END_RUNG
   RUNG wire#powerrail
      I_Contact( #FALSE )
      Not()
      Contact( "Unit1.Em4.ControlNodes".cm.Interlock.anodeAlignTableAxisY1.source.posAbsolute[4] )
      Move(in := 4, out1 => "Unit1.Em4.ControlNodes".cmAnodeAlignTableAxisY1.commands.selectSetPosition)
      Coil( "Unit1.Em4.ControlNodes".cm.axisCommand.anodeAlignTableAxisY1.posAbsolute[4] )
   END_RUNG
   // the same network as SCL:
   #"AnodeAlignTableAxisY1 Position_"[4](PosiNo := 4,   // "Position.LER_Axis"
                           Status := #unitStatus,
                           commands := "Unit1.Em4.HmiInterface".cmAnodeAlignTableAxisY1.commands,
                           interlockOk := "Unit1.Em4.ControlNodes".cm.Interlock.anodeAlignTableAxisY1.source.posAbsolute,
                           intOut := "Unit1.Em4.HmiInterface".intCondition.Axis_16.Position.intOut);
   #_w1 := NOT (NOT #FALSE) AND "Unit1.Em4.ControlNodes".cm.Interlock.anodeAlignTableAxisY1.source.posAbsolute[4];
   IF #_w1 THEN "Unit1.Em4.ControlNodes".cmAnodeAlignTableAxisY1.commands.selectSetPosition := 4; END_IF;
   "Unit1.Em4.ControlNodes".cm.axisCommand.anodeAlignTableAxisY1.posAbsolute[4] := #_w1;
END_REGION

REGION Network 192: CmAnodeAlignTableAxisY1 Position Absolute Position5
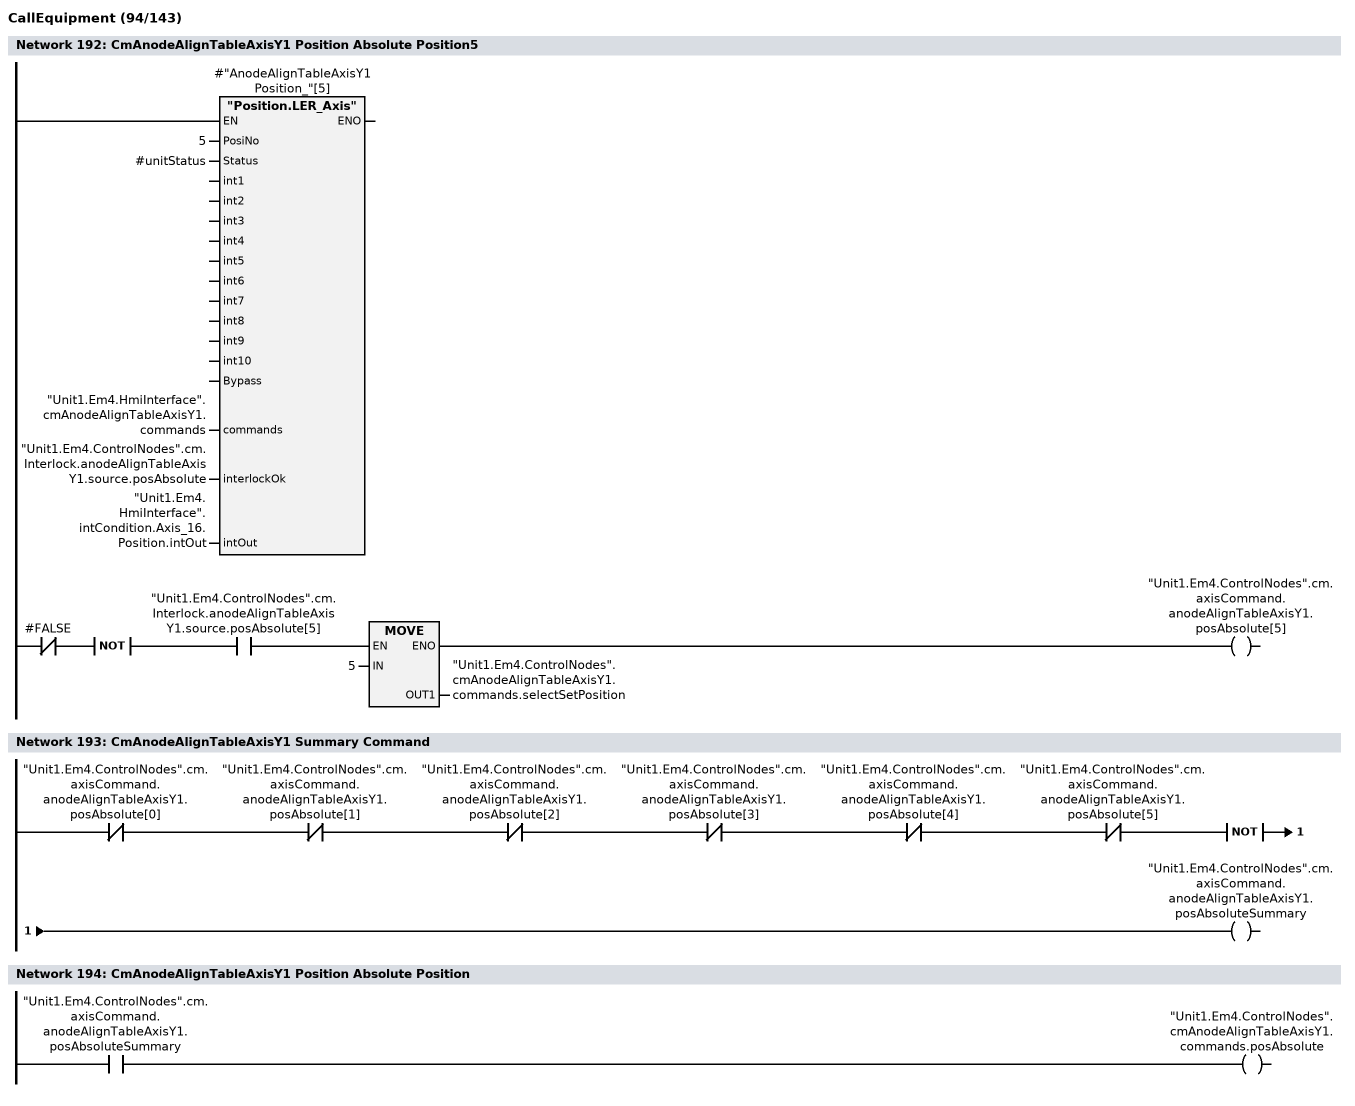
   RUNG wire#powerrail
      #"AnodeAlignTableAxisY1 Position_"[5](PosiNo := 5, Status := #unitStatus, int1 :=, int2 :=, int3 :=, int4 :=, int5 :=, int6 :=, int7 :=, int8 :=, int9 :=, int10 :=, Bypass :=, commands := "Unit1.Em4.HmiInterface".cmAnodeAlignTableAxisY1.commands, interlockOk := "Unit1.Em4.ControlNodes".cm.Interlock.anodeAlignTableAxisY1.source.posAbsolute, intOut := "Unit1.Em4.HmiInterface".intCondition.Axis_16.Position.intOut)
   END_RUNG
   RUNG wire#powerrail
      I_Contact( #FALSE )
      Not()
      Contact( "Unit1.Em4.ControlNodes".cm.Interlock.anodeAlignTableAxisY1.source.posAbsolute[5] )
      Move(in := 5, out1 => "Unit1.Em4.ControlNodes".cmAnodeAlignTableAxisY1.commands.selectSetPosition)
      Coil( "Unit1.Em4.ControlNodes".cm.axisCommand.anodeAlignTableAxisY1.posAbsolute[5] )
   END_RUNG
   // the same network as SCL:
   #"AnodeAlignTableAxisY1 Position_"[5](PosiNo := 5,   // "Position.LER_Axis"
                           Status := #unitStatus,
                           commands := "Unit1.Em4.HmiInterface".cmAnodeAlignTableAxisY1.commands,
                           interlockOk := "Unit1.Em4.ControlNodes".cm.Interlock.anodeAlignTableAxisY1.source.posAbsolute,
                           intOut := "Unit1.Em4.HmiInterface".intCondition.Axis_16.Position.intOut);
   #_w1 := NOT (NOT #FALSE) AND "Unit1.Em4.ControlNodes".cm.Interlock.anodeAlignTableAxisY1.source.posAbsolute[5];
   IF #_w1 THEN "Unit1.Em4.ControlNodes".cmAnodeAlignTableAxisY1.commands.selectSetPosition := 5; END_IF;
   "Unit1.Em4.ControlNodes".cm.axisCommand.anodeAlignTableAxisY1.posAbsolute[5] := #_w1;
END_REGION

REGION Network 193: CmAnodeAlignTableAxisY1 Summary Command
   RUNG wire#powerrail
      I_Contact( "Unit1.Em4.ControlNodes".cm.axisCommand.anodeAlignTableAxisY1.posAbsolute[0] )
      I_Contact( "Unit1.Em4.ControlNodes".cm.axisCommand.anodeAlignTableAxisY1.posAbsolute[1] )
      I_Contact( "Unit1.Em4.ControlNodes".cm.axisCommand.anodeAlignTableAxisY1.posAbsolute[2] )
      I_Contact( "Unit1.Em4.ControlNodes".cm.axisCommand.anodeAlignTableAxisY1.posAbsolute[3] )
      I_Contact( "Unit1.Em4.ControlNodes".cm.axisCommand.anodeAlignTableAxisY1.posAbsolute[4] )
      I_Contact( "Unit1.Em4.ControlNodes".cm.axisCommand.anodeAlignTableAxisY1.posAbsolute[5] )
      Not()
      Coil( "Unit1.Em4.ControlNodes".cm.axisCommand.anodeAlignTableAxisY1.posAbsoluteSummary )
   END_RUNG
   // the same network as SCL:
   "Unit1.Em4.ControlNodes".cm.axisCommand.anodeAlignTableAxisY1.posAbsoluteSummary := NOT (NOT "Unit1.Em4.ControlNodes".cm.axisCommand.anodeAlignTableAxisY1.posAbsolute[0] AND NOT "Unit1.Em4.ControlNodes".cm.axisCommand.anodeAlignTableAxisY1.posAbsolute[1] AND NOT "Unit1.Em4.ControlNodes".cm.axisCommand.anodeAlignTableAxisY1.posAbsolute[2] AND NOT "Unit1.Em4.ControlNodes".cm.axisCommand.anodeAlignTableAxisY1.posAbsolute[3] AND NOT "Unit1.Em4.ControlNodes".cm.axisCommand.anodeAlignTableAxisY1.posAbsolute[4] AND NOT "Unit1.Em4.ControlNodes".cm.axisCommand.anodeAlignTableAxisY1.posAbsolute[5]);
END_REGION

REGION Network 194: CmAnodeAlignTableAxisY1 Position Absolute Position
   RUNG wire#powerrail
      Contact( "Unit1.Em4.ControlNodes".cm.axisCommand.anodeAlignTableAxisY1.posAbsoluteSummary )
      Coil( "Unit1.Em4.ControlNodes".cmAnodeAlignTableAxisY1.commands.posAbsolute )
   END_RUNG
   // the same network as SCL:
   "Unit1.Em4.ControlNodes".cmAnodeAlignTableAxisY1.commands.posAbsolute := "Unit1.Em4.ControlNodes".cm.axisCommand.anodeAlignTableAxisY1.posAbsoluteSummary;
END_REGION

REGION Network 195: CmAnodeAlignTableAxisY1 Interlock Summary
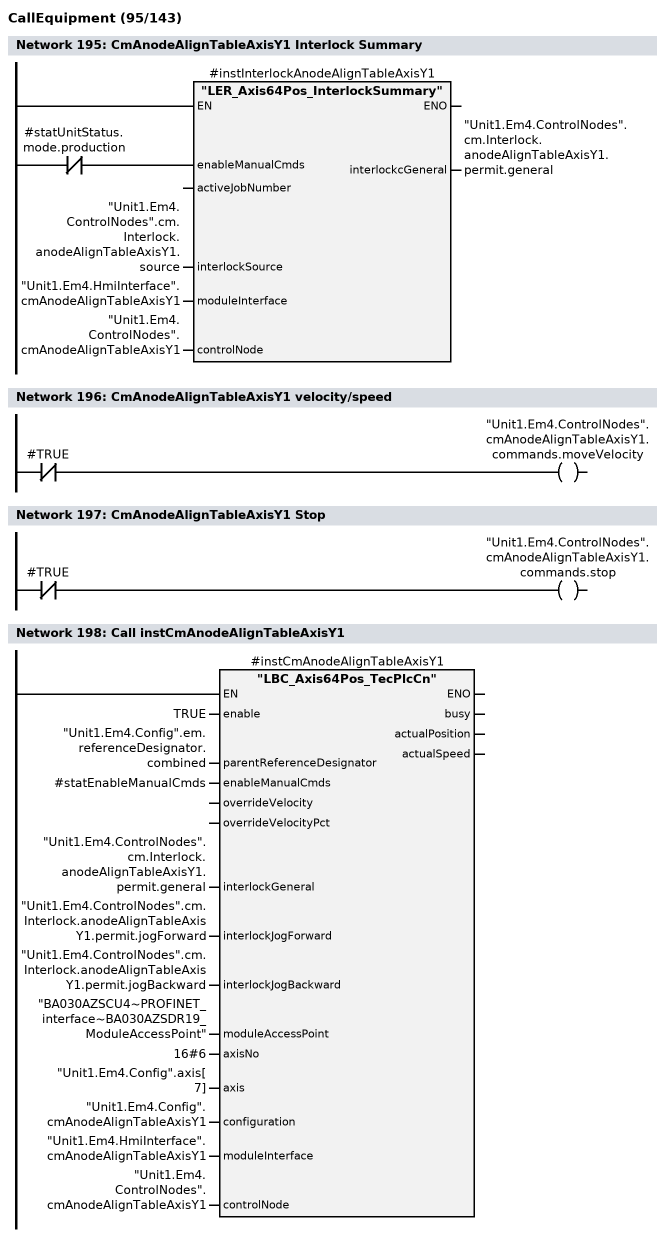
   RUNG wire#powerrail
      #instInterlockAnodeAlignTableAxisY1(enableManualCmds := wire#w1, activeJobNumber :=, interlockSource := "Unit1.Em4.ControlNodes".cm.Interlock.anodeAlignTableAxisY1.source, moduleInterface := "Unit1.Em4.HmiInterface".cmAnodeAlignTableAxisY1, controlNode := "Unit1.Em4.ControlNodes".cmAnodeAlignTableAxisY1, interlockcGeneral => "Unit1.Em4.ControlNodes".cm.Interlock.anodeAlignTableAxisY1.permit.general)
   END_RUNG
   RUNG wire#powerrail
      I_Contact( #statUnitStatus.mode.production )
   END_RUNG wire#w1
   // the same network as SCL:
   #instInterlockAnodeAlignTableAxisY1(enableManualCmds := NOT #statUnitStatus.mode.production,   // "LER_Axis64Pos_InterlockSummary"
                           interlockSource := "Unit1.Em4.ControlNodes".cm.Interlock.anodeAlignTableAxisY1.source,
                           moduleInterface := "Unit1.Em4.HmiInterface".cmAnodeAlignTableAxisY1,
                           controlNode := "Unit1.Em4.ControlNodes".cmAnodeAlignTableAxisY1,
                           interlockcGeneral => "Unit1.Em4.ControlNodes".cm.Interlock.anodeAlignTableAxisY1.permit.general);
END_REGION

REGION Network 196: CmAnodeAlignTableAxisY1 velocity/speed
   RUNG wire#powerrail
      I_Contact( #TRUE )
      Coil( "Unit1.Em4.ControlNodes".cmAnodeAlignTableAxisY1.commands.moveVelocity )
   END_RUNG
   // the same network as SCL:
   "Unit1.Em4.ControlNodes".cmAnodeAlignTableAxisY1.commands.moveVelocity := NOT #TRUE;
END_REGION

REGION Network 197: CmAnodeAlignTableAxisY1 Stop
   RUNG wire#powerrail
      I_Contact( #TRUE )
      Coil( "Unit1.Em4.ControlNodes".cmAnodeAlignTableAxisY1.commands.stop )
   END_RUNG
   // the same network as SCL:
   "Unit1.Em4.ControlNodes".cmAnodeAlignTableAxisY1.commands.stop := NOT #TRUE;
END_REGION

REGION Network 198: Call instCmAnodeAlignTableAxisY1
   RUNG wire#powerrail
      #instCmAnodeAlignTableAxisY1(enable := TRUE, parentReferenceDesignator := "Unit1.Em4.Config".em.referenceDesignator.combined, enableManualCmds := #statEnableManualCmds, overrideVelocity :=, overrideVelocityPct :=, interlockGeneral := "Unit1.Em4.ControlNodes".cm.Interlock.anodeAlignTableAxisY1.permit.general, interlockJogForward := "Unit1.Em4.ControlNodes".cm.Interlock.anodeAlignTableAxisY1.permit.jogForward, interlockJogBackward := "Unit1.Em4.ControlNodes".cm.Interlock.anodeAlignTableAxisY1.permit.jogBackward, moduleAccessPoint := "BA030AZSCU4~PROFINET_interface~BA030AZSDR19_ModuleAccessPoint", axisNo := 16#6, axis := "Unit1.Em4.Config".axis[7], configuration := "Unit1.Em4.Config".cmAnodeAlignTableAxisY1, moduleInterface := "Unit1.Em4.HmiInterface".cmAnodeAlignTableAxisY1, controlNode := "Unit1.Em4.ControlNodes".cmAnodeAlignTableAxisY1, busy =>, actualPosition =>, actualSpeed =>)
   END_RUNG
   // the same network as SCL:
   #instCmAnodeAlignTableAxisY1(enable := TRUE,   // "LBC_Axis64Pos_TecPlcCn"
                           parentReferenceDesignator := "Unit1.Em4.Config".em.referenceDesignator.combined,
                           enableManualCmds := #statEnableManualCmds,
                           interlockGeneral := "Unit1.Em4.ControlNodes".cm.Interlock.anodeAlignTableAxisY1.permit.general,
                           interlockJogForward := "Unit1.Em4.ControlNodes".cm.Interlock.anodeAlignTableAxisY1.permit.jogForward,
                           interlockJogBackward := "Unit1.Em4.ControlNodes".cm.Interlock.anodeAlignTableAxisY1.permit.jogBackward,
                           moduleAccessPoint := "BA030AZSCU4~PROFINET_interface~BA030AZSDR19_ModuleAccessPoint",
                           axisNo := 16#6,
                           axis := "Unit1.Em4.Config".axis[7],
                           configuration := "Unit1.Em4.Config".cmAnodeAlignTableAxisY1,
                           moduleInterface := "Unit1.Em4.HmiInterface".cmAnodeAlignTableAxisY1,
                           controlNode := "Unit1.Em4.ControlNodes".cmAnodeAlignTableAxisY1);
END_REGION

REGION Network 199: AnodeAlignTableAxisY1 SoftCam
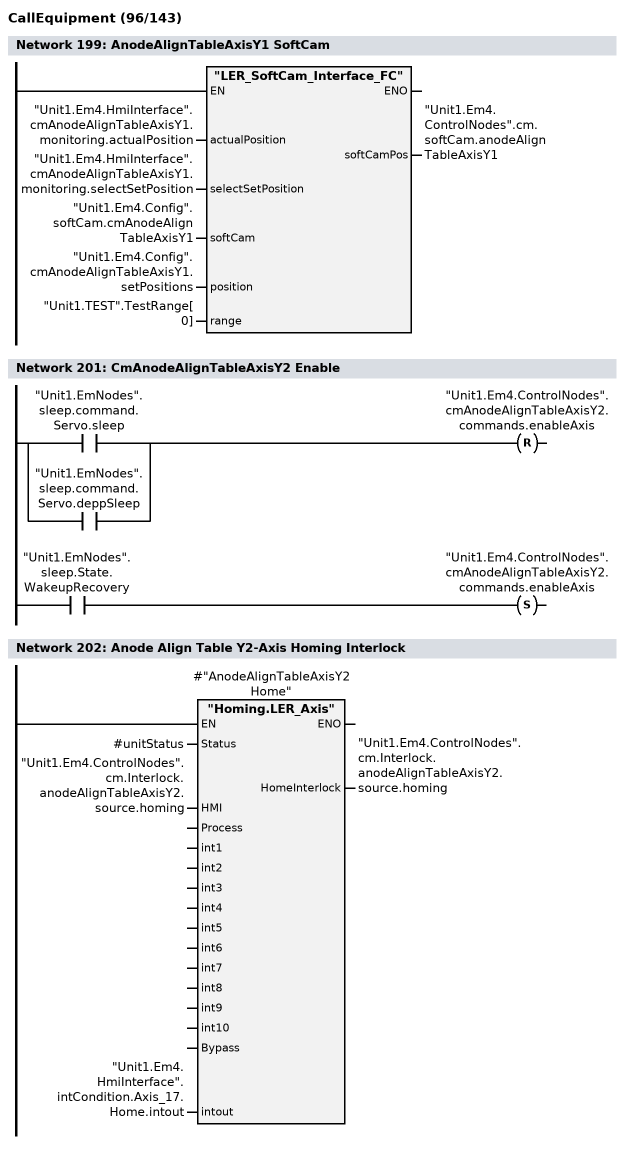
   RUNG wire#powerrail
      "LER_SoftCam_Interface_FC"(actualPosition := "Unit1.Em4.HmiInterface".cmAnodeAlignTableAxisY1.monitoring.actualPosition, selectSetPosition := "Unit1.Em4.HmiInterface".cmAnodeAlignTableAxisY1.monitoring.selectSetPosition, softCam := "Unit1.Em4.Config".softCam.cmAnodeAlignTableAxisY1, position := "Unit1.Em4.Config".cmAnodeAlignTableAxisY1.setPositions, range := "Unit1.TEST".TestRange[0], softCamPos => "Unit1.Em4.ControlNodes".cm.softCam.anodeAlignTableAxisY1)
   END_RUNG
   // the same network as SCL:
   "LER_SoftCam_Interface_FC"(actualPosition := "Unit1.Em4.HmiInterface".cmAnodeAlignTableAxisY1.monitoring.actualPosition,
                           selectSetPosition := "Unit1.Em4.HmiInterface".cmAnodeAlignTableAxisY1.monitoring.selectSetPosition,
                           softCam := "Unit1.Em4.Config".softCam.cmAnodeAlignTableAxisY1,
                           position := "Unit1.Em4.Config".cmAnodeAlignTableAxisY1.setPositions,
                           range := "Unit1.TEST".TestRange[0],
                           softCamPos => "Unit1.Em4.ControlNodes".cm.softCam.anodeAlignTableAxisY1);
END_REGION

REGION Network 201: CmAnodeAlignTableAxisY2 Enable
   RUNG wire#powerrail
      Contact( "Unit1.EmNodes".sleep.command.Servo.sleep )
      wire#w1
      R_Coil( "Unit1.Em4.ControlNodes".cmAnodeAlignTableAxisY2.commands.enableAxis )
   END_RUNG
   RUNG wire#powerrail
      Contact( "Unit1.EmNodes".sleep.command.Servo.deppSleep )
   END_RUNG wire#w1
   RUNG wire#powerrail
      Contact( "Unit1.EmNodes".sleep.State.WakeupRecovery )
      S_Coil( "Unit1.Em4.ControlNodes".cmAnodeAlignTableAxisY2.commands.enableAxis )
   END_RUNG
   // the same network as SCL:
   IF "Unit1.EmNodes".sleep.command.Servo.sleep OR "Unit1.EmNodes".sleep.command.Servo.deppSleep THEN
       "Unit1.Em4.ControlNodes".cmAnodeAlignTableAxisY2.commands.enableAxis := FALSE;
   END_IF;
   IF "Unit1.EmNodes".sleep.State.WakeupRecovery THEN
       "Unit1.Em4.ControlNodes".cmAnodeAlignTableAxisY2.commands.enableAxis := TRUE;
   END_IF;
END_REGION

REGION Network 202: Anode Align Table Y2-Axis Homing Interlock
   RUNG wire#powerrail
      #"AnodeAlignTableAxisY2 Home"(Status := #unitStatus, HMI := "Unit1.Em4.ControlNodes".cm.Interlock.anodeAlignTableAxisY2.source.homing, Process :=, int1 :=, int2 :=, int3 :=, int4 :=, int5 :=, int6 :=, int7 :=, int8 :=, int9 :=, int10 :=, Bypass :=, intout := "Unit1.Em4.HmiInterface".intCondition.Axis_17.Home.intout, HomeInterlock => "Unit1.Em4.ControlNodes".cm.Interlock.anodeAlignTableAxisY2.source.homing)
   END_RUNG
   // the same network as SCL:
   #"AnodeAlignTableAxisY2 Home"(Status := #unitStatus,   // "Homing.LER_Axis"
                           HMI := "Unit1.Em4.ControlNodes".cm.Interlock.anodeAlignTableAxisY2.source.homing,
                           intout := "Unit1.Em4.HmiInterface".intCondition.Axis_17.Home.intout,
                           HomeInterlock => "Unit1.Em4.ControlNodes".cm.Interlock.anodeAlignTableAxisY2.source.homing);
END_REGION

REGION Network 203: CmAnodeAlignTableAxisY2 Position Absolute Jog
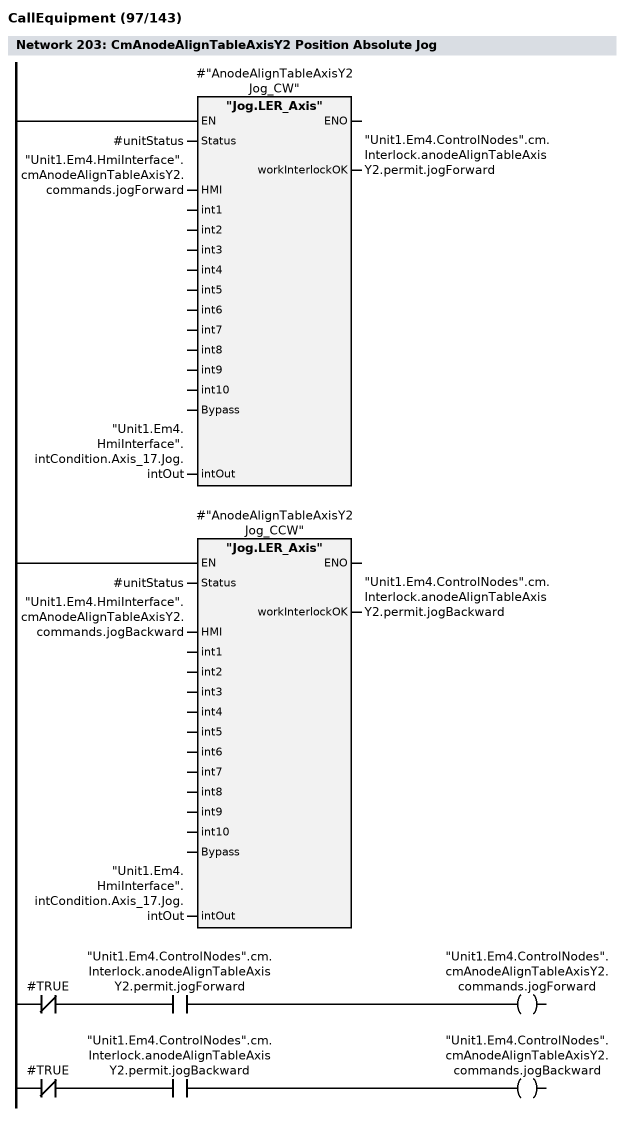
   RUNG wire#powerrail
      #"AnodeAlignTableAxisY2 Jog_CW"(Status := #unitStatus, HMI := "Unit1.Em4.HmiInterface".cmAnodeAlignTableAxisY2.commands.jogForward, int1 :=, int2 :=, int3 :=, int4 :=, int5 :=, int6 :=, int7 :=, int8 :=, int9 :=, int10 :=, Bypass :=, intOut := "Unit1.Em4.HmiInterface".intCondition.Axis_17.Jog.intOut, workInterlockOK => "Unit1.Em4.ControlNodes".cm.Interlock.anodeAlignTableAxisY2.permit.jogForward)
   END_RUNG
   RUNG wire#powerrail
      #"AnodeAlignTableAxisY2 Jog_CCW"(Status := #unitStatus, HMI := "Unit1.Em4.HmiInterface".cmAnodeAlignTableAxisY2.commands.jogBackward, int1 :=, int2 :=, int3 :=, int4 :=, int5 :=, int6 :=, int7 :=, int8 :=, int9 :=, int10 :=, Bypass :=, intOut := "Unit1.Em4.HmiInterface".intCondition.Axis_17.Jog.intOut, workInterlockOK => "Unit1.Em4.ControlNodes".cm.Interlock.anodeAlignTableAxisY2.permit.jogBackward)
   END_RUNG
   RUNG wire#powerrail
      I_Contact( #TRUE )
      Contact( "Unit1.Em4.ControlNodes".cm.Interlock.anodeAlignTableAxisY2.permit.jogForward )
      Coil( "Unit1.Em4.ControlNodes".cmAnodeAlignTableAxisY2.commands.jogForward )
   END_RUNG
   RUNG wire#powerrail
      I_Contact( #TRUE )
      Contact( "Unit1.Em4.ControlNodes".cm.Interlock.anodeAlignTableAxisY2.permit.jogBackward )
      Coil( "Unit1.Em4.ControlNodes".cmAnodeAlignTableAxisY2.commands.jogBackward )
   END_RUNG
   // the same network as SCL:
   #"AnodeAlignTableAxisY2 Jog_CW"(Status := #unitStatus,   // "Jog.LER_Axis"
                           HMI := "Unit1.Em4.HmiInterface".cmAnodeAlignTableAxisY2.commands.jogForward,
                           intOut := "Unit1.Em4.HmiInterface".intCondition.Axis_17.Jog.intOut,
                           workInterlockOK => "Unit1.Em4.ControlNodes".cm.Interlock.anodeAlignTableAxisY2.permit.jogForward);
   #"AnodeAlignTableAxisY2 Jog_CCW"(Status := #unitStatus,   // "Jog.LER_Axis"
                           HMI := "Unit1.Em4.HmiInterface".cmAnodeAlignTableAxisY2.commands.jogBackward,
                           intOut := "Unit1.Em4.HmiInterface".intCondition.Axis_17.Jog.intOut,
                           workInterlockOK => "Unit1.Em4.ControlNodes".cm.Interlock.anodeAlignTableAxisY2.permit.jogBackward);
   "Unit1.Em4.ControlNodes".cmAnodeAlignTableAxisY2.commands.jogForward := NOT #TRUE AND "Unit1.Em4.ControlNodes".cm.Interlock.anodeAlignTableAxisY2.permit.jogForward;
   "Unit1.Em4.ControlNodes".cmAnodeAlignTableAxisY2.commands.jogBackward := NOT #TRUE AND "Unit1.Em4.ControlNodes".cm.Interlock.anodeAlignTableAxisY2.permit.jogBackward;
END_REGION

REGION Network 204: CmAnodeAlignTableAxisY2 Position Absolute Position0
